Yaskawa INFORM job: DEMO_ROOF_UPPER_0625_3PAINT_63.JBI

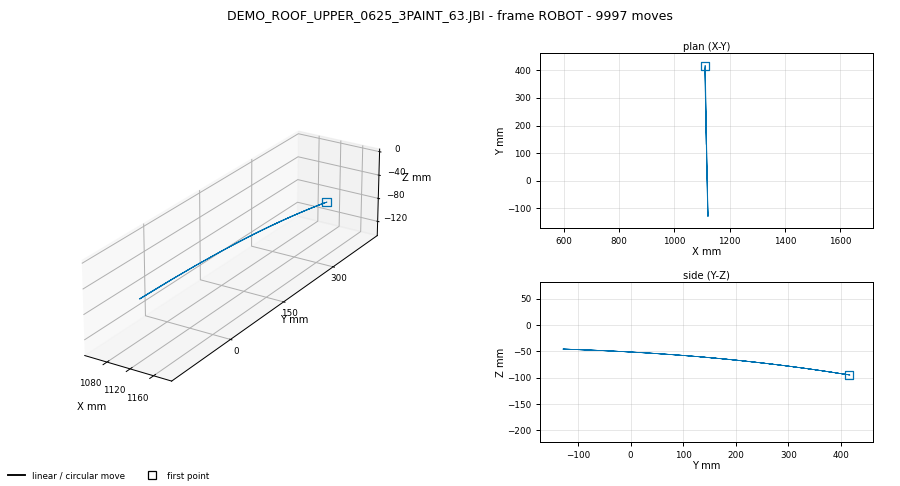
[picture p0: tool path of DEMO_ROOF_UPPER_0625_3PAINT_63.JBI in frame ROBOT, 9997 of 9997 moves have a stored position in this frame; points joined in program order, loops and branches not executed]
/JOB
//NAME DEMO_ROOF_UPPER_0625_3PAINT63
//POS
///NPOS 9997,0,0,0,0,0
///TOOL 0
///USER 0
///POSTYPE ROBOT
///RECTAN
///RCONF 1,0,0,0,0,0,0,0,0,0,0,0,0,0,0,0,0,0,0,0,0,0,0,0
C00000=1111.542,415.356,-94.503,-176.518,11.839,149.535
C00001=1111.541,415.109,-94.464,-176.519,11.832,149.534
C00002=1111.542,414.862,-94.424,-176.521,11.826,149.533
C00003=1111.542,414.615,-94.385,-176.522,11.820,149.532
C00004=1111.543,414.368,-94.345,-176.524,11.814,149.530
C00005=1111.545,414.121,-94.306,-176.526,11.807,149.529
C00006=1111.547,413.875,-94.266,-176.528,11.801,149.528
C00007=1111.549,413.627,-94.227,-176.529,11.795,149.527
C00008=1111.553,413.381,-94.187,-176.531,11.789,149.526
C00009=1111.556,413.135,-94.147,-176.533,11.783,149.525
C00010=1111.560,412.887,-94.107,-176.535,11.777,149.523
C00011=1111.563,412.640,-94.067,-176.536,11.771,149.522
C00012=1111.567,412.393,-94.027,-176.538,11.765,149.521
C00013=1111.570,412.147,-93.987,-176.540,11.759,149.520
C00014=1111.574,411.900,-93.948,-176.542,11.754,149.519
C00015=1111.577,411.654,-93.908,-176.543,11.747,149.518
C00016=1111.580,411.407,-93.869,-176.546,11.741,149.517
C00017=1111.584,411.160,-93.830,-176.547,11.736,149.516
C00018=1111.588,410.913,-93.789,-176.549,11.730,149.515
C00019=1111.591,410.666,-93.750,-176.551,11.725,149.514
C00020=1111.594,410.419,-93.710,-176.553,11.719,149.513
C00021=1111.598,410.172,-93.670,-176.554,11.713,149.512
C00022=1111.602,409.925,-93.631,-176.557,11.707,149.511
C00023=1111.605,409.679,-93.591,-176.559,11.703,149.510
C00024=1111.609,409.432,-93.552,-176.561,11.697,149.509
C00025=1111.612,409.185,-93.513,-176.562,11.691,149.508
C00026=1111.616,408.938,-93.473,-176.564,11.686,149.507
C00027=1111.619,408.692,-93.433,-176.567,11.680,149.506
C00028=1111.623,408.445,-93.394,-176.568,11.675,149.505
C00029=1111.626,408.198,-93.355,-176.570,11.670,149.504
C00030=1111.630,407.951,-93.316,-176.572,11.664,149.503
C00031=1111.633,407.704,-93.276,-176.574,11.659,149.503
C00032=1111.637,407.458,-93.236,-176.576,11.654,149.502
C00033=1111.641,407.211,-93.197,-176.578,11.649,149.501
C00034=1111.644,406.964,-93.158,-176.580,11.644,149.500
C00035=1111.648,406.717,-93.119,-176.582,11.639,149.499
C00036=1111.651,406.470,-93.079,-176.584,11.634,149.498
C00037=1111.654,406.223,-93.041,-176.586,11.629,149.498
C00038=1111.658,405.976,-93.002,-176.588,11.624,149.497
C00039=1111.662,405.729,-92.962,-176.590,11.619,149.496
C00040=1111.665,405.483,-92.922,-176.592,11.614,149.495
C00041=1111.668,405.236,-92.883,-176.594,11.609,149.494
C00042=1111.672,404.989,-92.844,-176.596,11.604,149.494
C00043=1111.676,404.742,-92.805,-176.599,11.599,149.493
C00044=1111.679,404.495,-92.765,-176.601,11.594,149.492
C00045=1111.682,404.248,-92.727,-176.603,11.590,149.492
C00046=1111.686,404.001,-92.687,-176.605,11.585,149.491
C00047=1111.690,403.754,-92.649,-176.607,11.581,149.490
C00048=1111.693,403.543,-92.615,-176.609,11.576,149.490
C00049=1111.696,403.331,-92.582,-176.611,11.572,149.489
C00050=1111.699,403.121,-92.548,-176.613,11.569,149.488
C00051=1111.702,402.909,-92.515,-176.615,11.565,149.488
C00052=1111.705,402.697,-92.482,-176.616,11.561,149.487
C00053=1111.708,402.486,-92.448,-176.619,11.556,149.487
C00054=1111.711,402.275,-92.415,-176.620,11.553,149.486
C00055=1111.714,402.063,-92.381,-176.622,11.549,149.486
C00056=1111.718,401.817,-92.342,-176.624,11.544,149.485
C00057=1111.721,401.570,-92.304,-176.626,11.541,149.484
C00058=1111.725,401.323,-92.264,-176.628,11.536,149.484
C00059=1111.729,401.075,-92.226,-176.631,11.532,149.483
C00060=1111.732,400.828,-92.187,-176.634,11.527,149.483
C00061=1111.735,400.582,-92.148,-176.635,11.523,149.482
C00062=1111.739,400.335,-92.109,-176.638,11.519,149.482
C00063=1111.743,400.087,-92.070,-176.640,11.514,149.481
C00064=1111.746,399.841,-92.032,-176.642,11.511,149.481
C00065=1111.750,399.594,-91.993,-176.645,11.506,149.480
C00066=1111.753,399.347,-91.953,-176.647,11.502,149.480
C00067=1111.757,399.100,-91.916,-176.649,11.498,149.479
C00068=1111.760,398.853,-91.876,-176.652,11.494,149.479
C00069=1111.764,398.606,-91.838,-176.654,11.490,149.478
C00070=1111.768,398.360,-91.799,-176.656,11.486,149.478
C00071=1111.771,398.113,-91.760,-176.658,11.482,149.477
C00072=1111.775,397.865,-91.722,-176.661,11.478,149.477
C00073=1111.778,397.618,-91.683,-176.663,11.475,149.477
C00074=1111.782,397.371,-91.644,-176.666,11.470,149.476
C00075=1111.786,397.125,-91.606,-176.668,11.467,149.476
C00076=1111.789,396.877,-91.568,-176.671,11.463,149.475
C00077=1111.793,396.630,-91.528,-176.673,11.459,149.475
C00078=1111.796,396.383,-91.490,-176.675,11.456,149.475
C00079=1111.800,396.137,-91.452,-176.678,11.451,149.474
C00080=1111.804,395.890,-91.414,-176.680,11.448,149.474
C00081=1111.807,395.643,-91.374,-176.682,11.444,149.473
C00082=1111.811,395.395,-91.336,-176.685,11.440,149.473
C00083=1111.815,395.149,-91.298,-176.687,11.437,149.473
C00084=1111.819,394.902,-91.259,-176.689,11.433,149.472
C00085=1111.821,394.655,-91.220,-176.692,11.430,149.472
C00086=1111.825,394.407,-91.182,-176.694,11.426,149.472
C00087=1111.829,394.161,-91.144,-176.697,11.423,149.472
C00088=1111.833,393.914,-91.105,-176.699,11.419,149.471
C00089=1111.836,393.666,-91.067,-176.702,11.416,149.471
C00090=1111.841,393.420,-91.029,-176.704,11.412,149.471
C00091=1111.843,393.173,-90.990,-176.707,11.409,149.471
C00092=1111.847,392.925,-90.952,-176.709,11.406,149.470
C00093=1111.851,392.679,-90.914,-176.711,11.402,149.470
C00094=1111.855,392.431,-90.876,-176.714,11.398,149.470
C00095=1111.858,392.185,-90.837,-176.717,11.395,149.470
C00096=1111.862,391.937,-90.798,-176.719,11.392,149.469
C00097=1111.866,391.690,-90.761,-176.722,11.389,149.469
C00098=1111.869,391.443,-90.723,-176.724,11.386,149.469
C00099=1111.872,391.196,-90.684,-176.727,11.383,149.469
C00100=1111.876,390.950,-90.646,-176.729,11.379,149.469
C00101=1111.880,390.702,-90.608,-176.732,11.376,149.468
C00102=1111.883,390.455,-90.570,-176.734,11.373,149.468
C00103=1111.887,390.208,-90.532,-176.737,11.370,149.468
C00104=1111.890,389.996,-90.499,-176.739,11.368,149.468
C00105=1111.893,389.786,-90.466,-176.742,11.365,149.468
C00106=1111.897,389.573,-90.434,-176.744,11.363,149.468
C00107=1111.899,389.362,-90.401,-176.746,11.359,149.468
C00108=1111.903,389.151,-90.368,-176.748,11.357,149.468
C00109=1111.906,388.939,-90.336,-176.750,11.355,149.468
C00110=1111.910,388.728,-90.303,-176.753,11.352,149.467
C00111=1111.912,388.517,-90.271,-176.755,11.349,149.467
C00112=1111.915,388.269,-90.233,-176.757,11.347,149.467
C00113=1111.920,388.022,-90.194,-176.760,11.344,149.467
C00114=1111.923,387.775,-90.156,-176.762,11.341,149.467
C00115=1111.927,387.529,-90.119,-176.765,11.339,149.467
C00116=1111.931,387.281,-90.080,-176.768,11.336,149.467
C00117=1111.934,387.034,-90.042,-176.770,11.333,149.467
C00118=1111.938,386.787,-90.005,-176.773,11.330,149.467
C00119=1111.941,386.540,-89.967,-176.775,11.328,149.467
C00120=1111.945,386.293,-89.929,-176.778,11.325,149.467
C00121=1111.949,386.045,-89.892,-176.781,11.322,149.467
C00122=1111.953,385.799,-89.854,-176.784,11.319,149.467
C00123=1111.956,385.551,-89.816,-176.786,11.317,149.467
C00124=1111.960,385.304,-89.777,-176.789,11.314,149.467
C00125=1111.963,385.057,-89.740,-176.792,11.311,149.467
C00126=1111.967,384.810,-89.702,-176.794,11.309,149.467
C00127=1111.970,384.563,-89.664,-176.797,11.306,149.467
C00128=1111.974,384.316,-89.626,-176.800,11.303,149.467
C00129=1111.978,384.069,-89.589,-176.802,11.301,149.467
C00130=1111.982,383.821,-89.551,-176.805,11.299,149.467
C00131=1111.985,383.575,-89.513,-176.808,11.296,149.467
C00132=1111.989,383.327,-89.476,-176.810,11.294,149.467
C00133=1111.992,383.081,-89.438,-176.814,11.290,149.467
C00134=1111.996,382.833,-89.401,-176.817,11.288,149.467
C00135=1112.000,382.586,-89.363,-176.820,11.285,149.467
C00136=1112.004,382.339,-89.325,-176.823,11.283,149.467
C00137=1112.008,382.092,-89.288,-176.827,11.280,149.468
C00138=1112.011,381.844,-89.250,-176.830,11.278,149.468
C00139=1112.015,381.598,-89.212,-176.833,11.275,149.468
C00140=1112.018,381.350,-89.175,-176.836,11.272,149.468
C00141=1112.022,381.103,-89.137,-176.840,11.269,149.468
C00142=1112.026,380.857,-89.100,-176.843,11.266,149.468
C00143=1112.029,380.609,-89.063,-176.846,11.264,149.468
C00144=1112.034,380.362,-89.024,-176.850,11.261,149.469
C00145=1112.037,380.115,-88.987,-176.853,11.259,149.469
C00146=1112.041,379.868,-88.950,-176.856,11.256,149.469
C00147=1112.044,379.620,-88.912,-176.859,11.253,149.469
C00148=1112.048,379.373,-88.875,-176.862,11.251,149.469
C00149=1112.052,379.127,-88.837,-176.866,11.249,149.469
C00150=1112.056,378.879,-88.800,-176.869,11.246,149.469
C00151=1112.059,378.632,-88.763,-176.872,11.242,149.470
C00152=1112.063,378.384,-88.725,-176.876,11.240,149.470
C00153=1112.067,378.138,-88.688,-176.879,11.237,149.470
C00154=1112.071,377.890,-88.651,-176.882,11.235,149.470
C00155=1112.074,377.643,-88.613,-176.886,11.232,149.470
C00156=1112.078,377.396,-88.576,-176.889,11.230,149.471
C00157=1112.082,377.149,-88.539,-176.892,11.228,149.471
C00158=1112.085,376.901,-88.501,-176.895,11.225,149.471
C00159=1112.089,376.654,-88.464,-176.898,11.222,149.471
C00160=1112.092,376.442,-88.432,-176.902,11.220,149.471
C00161=1112.095,376.231,-88.401,-176.904,11.218,149.471
C00162=1112.099,376.020,-88.369,-176.907,11.216,149.471
C00163=1112.102,375.808,-88.337,-176.910,11.214,149.472
C00164=1112.105,375.596,-88.306,-176.913,11.212,149.472
C00165=1112.108,375.385,-88.274,-176.915,11.209,149.472
C00166=1112.111,375.173,-88.242,-176.918,11.207,149.472
C00167=1112.114,374.962,-88.210,-176.921,11.205,149.472
C00168=1112.118,374.714,-88.173,-176.925,11.202,149.473
C00169=1112.122,374.467,-88.136,-176.928,11.200,149.473
C00170=1112.126,374.220,-88.099,-176.931,11.197,149.473
C00171=1112.130,373.973,-88.062,-176.935,11.195,149.473
C00172=1112.133,373.725,-88.025,-176.938,11.192,149.473
C00173=1112.137,373.478,-87.988,-176.941,11.190,149.474
C00174=1112.141,373.231,-87.951,-176.945,11.187,149.474
C00175=1112.144,372.983,-87.914,-176.948,11.185,149.474
C00176=1112.148,372.736,-87.877,-176.951,11.183,149.474
C00177=1112.152,372.489,-87.840,-176.954,11.180,149.474
C00178=1112.155,372.242,-87.804,-176.958,11.178,149.475
C00179=1112.159,371.994,-87.766,-176.961,11.175,149.475
C00180=1112.163,371.747,-87.729,-176.964,11.173,149.475
C00181=1112.167,371.500,-87.693,-176.968,11.170,149.475
C00182=1112.171,371.253,-87.656,-176.971,11.168,149.475
C00183=1112.174,371.005,-87.619,-176.975,11.165,149.476
C00184=1112.178,370.758,-87.582,-176.978,11.163,149.476
C00185=1112.182,370.511,-87.545,-176.981,11.161,149.476
C00186=1112.186,370.264,-87.509,-176.984,11.158,149.476
C00187=1112.190,370.017,-87.472,-176.988,11.156,149.477
C00188=1112.193,369.769,-87.435,-176.991,11.153,149.477
C00189=1112.196,369.522,-87.399,-176.994,11.151,149.477
C00190=1112.201,369.275,-87.362,-176.998,11.148,149.477
C00191=1112.205,369.028,-87.325,-177.001,11.146,149.478
C00192=1112.208,368.781,-87.289,-177.005,11.144,149.478
C00193=1112.212,368.533,-87.252,-177.008,11.141,149.478
C00194=1112.216,368.286,-87.215,-177.011,11.139,149.478
C00195=1112.219,368.038,-87.179,-177.015,11.136,149.478
C00196=1112.223,367.791,-87.142,-177.018,11.134,149.479
C00197=1112.227,367.544,-87.106,-177.022,11.131,149.479
C00198=1112.231,367.297,-87.069,-177.025,11.129,149.479
C00199=1112.235,367.050,-87.032,-177.028,11.127,149.480
C00200=1112.238,366.802,-86.996,-177.031,11.124,149.480
C00201=1112.242,366.554,-86.960,-177.035,11.122,149.480
C00202=1112.245,366.307,-86.923,-177.038,11.119,149.480
C00203=1112.250,366.060,-86.886,-177.042,11.117,149.481
C00204=1112.253,365.813,-86.851,-177.045,11.114,149.481
C00205=1112.257,365.566,-86.814,-177.048,11.112,149.481
C00206=1112.261,365.319,-86.778,-177.052,11.110,149.481
C00207=1112.265,365.071,-86.742,-177.055,11.107,149.482
C00208=1112.269,364.824,-86.705,-177.059,11.105,149.482
C00209=1112.272,364.576,-86.668,-177.062,11.102,149.482
C00210=1112.276,364.328,-86.632,-177.065,11.100,149.482
C00211=1112.280,364.081,-86.596,-177.069,11.097,149.482
C00212=1112.283,363.835,-86.559,-177.072,11.095,149.483
C00213=1112.287,363.587,-86.523,-177.075,11.094,149.483
C00214=1112.291,363.340,-86.487,-177.078,11.091,149.483
C00215=1112.295,363.092,-86.451,-177.082,11.089,149.483
C00216=1112.298,362.881,-86.420,-177.085,11.086,149.484
C00217=1112.301,362.669,-86.389,-177.088,11.085,149.484
C00218=1112.304,362.456,-86.358,-177.091,11.082,149.484
C00219=1112.307,362.245,-86.327,-177.094,11.080,149.484
C00220=1112.311,362.034,-86.296,-177.096,11.079,149.485
C00221=1112.314,361.822,-86.265,-177.100,11.076,149.485
C00222=1112.318,361.610,-86.234,-177.102,11.075,149.485
C00223=1112.321,361.398,-86.204,-177.105,11.072,149.485
C00224=1112.325,361.151,-86.167,-177.109,11.070,149.486
C00225=1112.329,360.903,-86.131,-177.112,11.067,149.486
C00226=1112.332,360.656,-86.095,-177.115,11.065,149.486
C00227=1112.336,360.409,-86.059,-177.119,11.062,149.486
C00228=1112.340,360.161,-86.023,-177.122,11.060,149.486
C00229=1112.343,359.914,-85.987,-177.126,11.058,149.487
C00230=1112.348,359.666,-85.951,-177.129,11.055,149.487
C00231=1112.351,359.419,-85.915,-177.132,11.053,149.487
C00232=1112.355,359.172,-85.879,-177.135,11.051,149.488
C00233=1112.359,358.925,-85.844,-177.138,11.048,149.488
C00234=1112.363,358.677,-85.807,-177.142,11.046,149.488
C00235=1112.366,358.430,-85.771,-177.145,11.044,149.488
C00236=1112.370,358.182,-85.736,-177.149,11.041,149.489
C00237=1112.374,357.935,-85.700,-177.152,11.039,149.489
C00238=1112.378,357.687,-85.664,-177.155,11.036,149.489
C00239=1112.381,357.440,-85.628,-177.159,11.034,149.489
C00240=1112.385,357.193,-85.592,-177.162,11.032,149.490
C00241=1112.389,356.945,-85.557,-177.166,11.029,149.490
C00242=1112.393,356.697,-85.520,-177.169,11.027,149.490
C00243=1112.397,356.450,-85.485,-177.172,11.024,149.490
C00244=1112.400,356.203,-85.449,-177.175,11.022,149.491
C00245=1112.404,355.956,-85.413,-177.179,11.020,149.491
C00246=1112.408,355.709,-85.378,-177.182,11.017,149.491
C00247=1112.412,355.461,-85.342,-177.186,11.015,149.491
C00248=1112.416,355.213,-85.306,-177.189,11.012,149.492
C00249=1112.420,354.966,-85.271,-177.192,11.010,149.492
C00250=1112.423,354.718,-85.235,-177.196,11.008,149.492
C00251=1112.427,354.471,-85.199,-177.199,11.005,149.492
C00252=1112.431,354.223,-85.164,-177.202,11.003,149.492
C00253=1112.435,353.977,-85.129,-177.206,11.000,149.493
C00254=1112.439,353.729,-85.093,-177.209,10.998,149.493
C00255=1112.442,353.482,-85.058,-177.213,10.996,149.493
C00256=1112.447,353.234,-85.022,-177.216,10.993,149.494
C00257=1112.450,352.986,-84.986,-177.219,10.991,149.494
C00258=1112.454,352.739,-84.950,-177.223,10.987,149.494
C00259=1112.458,352.492,-84.915,-177.227,10.985,149.494
C00260=1112.462,352.244,-84.880,-177.230,10.982,149.494
C00261=1112.466,351.997,-84.844,-177.233,10.980,149.495
C00262=1112.469,351.749,-84.809,-177.236,10.978,149.495
C00263=1112.473,351.501,-84.774,-177.240,10.975,149.495
C00264=1112.478,351.255,-84.739,-177.243,10.973,149.495
C00265=1112.481,351.007,-84.703,-177.246,10.970,149.496
C00266=1112.485,350.760,-84.667,-177.250,10.968,149.496
C00267=1112.489,350.512,-84.632,-177.253,10.965,149.496
C00268=1112.492,350.264,-84.597,-177.256,10.963,149.496
C00269=1112.497,350.017,-84.562,-177.260,10.960,149.496
C00270=1112.500,349.770,-84.526,-177.263,10.958,149.497
C00271=1112.504,349.522,-84.491,-177.266,10.955,149.497
C00272=1112.507,349.310,-84.461,-177.269,10.954,149.497
C00273=1112.511,349.098,-84.430,-177.272,10.951,149.497
C00274=1112.514,348.886,-84.401,-177.275,10.949,149.497
C00275=1112.518,348.675,-84.371,-177.277,10.948,149.498
C00276=1112.521,348.462,-84.341,-177.280,10.945,149.498
C00277=1112.525,348.251,-84.310,-177.283,10.943,149.498
C00278=1112.528,348.038,-84.281,-177.285,10.941,149.498
C00279=1112.531,347.827,-84.250,-177.288,10.939,149.498
C00280=1112.534,347.579,-84.215,-177.292,10.936,149.499
C00281=1112.538,347.331,-84.180,-177.295,10.934,149.499
C00282=1112.543,347.084,-84.145,-177.298,10.931,149.499
C00283=1112.547,346.836,-84.110,-177.301,10.929,149.499
C00284=1112.550,346.589,-84.074,-177.304,10.927,149.499
C00285=1112.555,346.341,-84.040,-177.307,10.924,149.500
C00286=1112.558,346.094,-84.005,-177.311,10.922,149.500
C00287=1112.561,345.847,-83.969,-177.314,10.919,149.500
C00288=1112.566,345.599,-83.935,-177.317,10.917,149.500
C00289=1112.570,345.352,-83.899,-177.320,10.914,149.500
C00290=1112.574,345.103,-83.865,-177.323,10.912,149.500
C00291=1112.578,344.856,-83.830,-177.327,10.909,149.501
C00292=1112.581,344.609,-83.795,-177.330,10.907,149.501
C00293=1112.586,344.361,-83.761,-177.332,10.905,149.501
C00294=1112.589,344.114,-83.725,-177.336,10.902,149.501
C00295=1112.593,343.866,-83.690,-177.339,10.900,149.501
C00296=1112.597,343.619,-83.656,-177.342,10.897,149.502
C00297=1112.601,343.371,-83.621,-177.346,10.895,149.502
C00298=1112.605,343.124,-83.586,-177.348,10.892,149.502
C00299=1112.609,342.876,-83.551,-177.352,10.890,149.502
C00300=1112.612,342.628,-83.517,-177.355,10.887,149.502
C00301=1112.617,342.381,-83.482,-177.358,10.885,149.503
C00302=1112.620,342.134,-83.447,-177.362,10.882,149.503
C00303=1112.625,341.886,-83.412,-177.365,10.879,149.503
C00304=1112.628,341.638,-83.378,-177.367,10.878,149.503
C00305=1112.633,341.391,-83.343,-177.371,10.875,149.503
C00306=1112.636,341.143,-83.308,-177.374,10.873,149.504
C00307=1112.640,340.896,-83.274,-177.377,10.870,149.504
C00308=1112.644,340.648,-83.239,-177.380,10.868,149.504
C00309=1112.648,340.400,-83.204,-177.384,10.865,149.504
C00310=1112.652,340.154,-83.170,-177.387,10.863,149.504
C00311=1112.656,339.905,-83.135,-177.390,10.860,149.505
C00312=1112.660,339.658,-83.101,-177.393,10.857,149.505
C00313=1112.664,339.410,-83.066,-177.396,10.855,149.505
C00314=1112.668,339.163,-83.032,-177.399,10.853,149.505
C00315=1112.671,338.915,-82.998,-177.402,10.851,149.505
C00316=1112.676,338.668,-82.963,-177.405,10.848,149.506
C00317=1112.680,338.419,-82.928,-177.409,10.846,149.506
C00318=1112.683,338.173,-82.894,-177.412,10.843,149.506
C00319=1112.687,337.925,-82.859,-177.415,10.841,149.506
C00320=1112.691,337.678,-82.825,-177.418,10.838,149.506
C00321=1112.695,337.430,-82.790,-177.421,10.836,149.506
C00322=1112.699,337.183,-82.756,-177.425,10.833,149.507
C00323=1112.703,336.934,-82.721,-177.428,10.831,149.507
C00324=1112.707,336.687,-82.688,-177.431,10.828,149.507
C00325=1112.711,336.439,-82.653,-177.434,10.826,149.507
C00326=1112.715,336.192,-82.619,-177.437,10.824,149.508
C00327=1112.719,335.945,-82.584,-177.440,10.821,149.508
C00328=1112.722,335.732,-82.555,-177.443,10.818,149.508
C00329=1112.726,335.519,-82.526,-177.446,10.817,149.508
C00330=1112.729,335.307,-82.496,-177.448,10.815,149.508
C00331=1112.732,335.096,-82.468,-177.452,10.812,149.508
C00332=1112.735,334.884,-82.438,-177.454,10.810,149.508
C00333=1112.739,334.672,-82.408,-177.457,10.809,149.509
C00334=1112.742,334.460,-82.379,-177.459,10.806,149.509
C00335=1112.746,334.247,-82.350,-177.462,10.804,149.509
C00336=1112.750,334.000,-82.317,-177.465,10.801,149.509
C00337=1112.754,333.752,-82.282,-177.468,10.799,149.509
C00338=1112.758,333.505,-82.248,-177.472,10.796,149.510
C00339=1112.762,333.257,-82.213,-177.475,10.794,149.510
C00340=1112.765,333.010,-82.179,-177.478,10.791,149.510
C00341=1112.769,332.762,-82.146,-177.481,10.790,149.510
C00342=1112.773,332.514,-82.111,-177.484,10.787,149.510
C00343=1112.777,332.267,-82.077,-177.487,10.784,149.510
C00344=1112.781,332.019,-82.043,-177.490,10.782,149.511
C00345=1112.785,331.771,-82.009,-177.494,10.779,149.511
C00346=1112.789,331.524,-81.975,-177.496,10.777,149.511
C00347=1112.792,331.276,-81.941,-177.500,10.774,149.511
C00348=1112.797,331.028,-81.907,-177.503,10.772,149.511
C00349=1112.801,330.781,-81.874,-177.506,10.769,149.512
C00350=1112.804,330.533,-81.839,-177.509,10.767,149.512
C00351=1112.809,330.285,-81.806,-177.513,10.764,149.512
C00352=1112.813,330.038,-81.772,-177.515,10.762,149.512
C00353=1112.817,329.789,-81.738,-177.518,10.760,149.512
C00354=1112.820,329.542,-81.704,-177.522,10.757,149.513
C00355=1112.825,329.295,-81.670,-177.525,10.755,149.513
C00356=1112.829,329.046,-81.636,-177.528,10.752,149.513
C00357=1112.832,328.799,-81.602,-177.531,10.750,149.513
C00358=1112.837,328.551,-81.569,-177.534,10.747,149.513
C00359=1112.840,328.304,-81.535,-177.537,10.744,149.513
C00360=1112.845,328.056,-81.501,-177.541,10.742,149.514
C00361=1112.848,327.808,-81.467,-177.544,10.739,149.514
C00362=1112.853,327.561,-81.434,-177.547,10.737,149.514
C00363=1112.856,327.313,-81.400,-177.550,10.735,149.514
C00364=1112.860,327.065,-81.367,-177.553,10.732,149.515
C00365=1112.865,326.818,-81.332,-177.556,10.730,149.515
C00366=1112.869,326.570,-81.299,-177.559,10.727,149.515
C00367=1112.872,326.322,-81.266,-177.563,10.725,149.515
C00368=1112.876,326.075,-81.232,-177.565,10.722,149.515
C00369=1112.880,325.827,-81.199,-177.569,10.720,149.515
C00370=1112.884,325.579,-81.166,-177.572,10.717,149.516
C00371=1112.888,325.332,-81.132,-177.575,10.714,149.516
C00372=1112.892,325.084,-81.098,-177.578,10.712,149.516
C00373=1112.897,324.835,-81.064,-177.581,10.710,149.516
C00374=1112.900,324.588,-81.030,-177.584,10.707,149.516
C00375=1112.905,324.341,-80.997,-177.587,10.705,149.517
C00376=1112.908,324.092,-80.964,-177.591,10.703,149.517
C00377=1112.912,323.845,-80.930,-177.593,10.700,149.517
C00378=1112.916,323.597,-80.897,-177.597,10.697,149.517
C00379=1112.920,323.350,-80.864,-177.600,10.695,149.517
C00380=1112.924,323.102,-80.830,-177.603,10.692,149.517
C00381=1112.928,322.854,-80.797,-177.606,10.690,149.518
C00382=1112.932,322.606,-80.763,-177.609,10.687,149.518
C00383=1112.936,322.359,-80.730,-177.613,10.684,149.518
C00384=1112.939,322.147,-80.702,-177.615,10.682,149.518
C00385=1112.943,321.934,-80.673,-177.618,10.681,149.518
C00386=1112.946,321.722,-80.645,-177.621,10.678,149.518
C00387=1112.949,321.510,-80.616,-177.623,10.676,149.519
C00388=1112.953,321.298,-80.588,-177.626,10.674,149.519
C00389=1112.956,321.085,-80.559,-177.628,10.672,149.519
C00390=1112.960,320.873,-80.531,-177.631,10.670,149.519
C00391=1112.963,320.660,-80.502,-177.633,10.668,149.519
C00392=1112.967,320.413,-80.469,-177.637,10.665,149.519
C00393=1112.971,320.165,-80.436,-177.640,10.663,149.520
C00394=1112.975,319.917,-80.403,-177.643,10.660,149.520
C00395=1112.979,319.670,-80.370,-177.646,10.658,149.520
C00396=1112.983,319.422,-80.337,-177.649,10.655,149.520
C00397=1112.987,319.174,-80.304,-177.653,10.653,149.520
C00398=1112.991,318.927,-80.270,-177.656,10.650,149.521
C00399=1112.995,318.678,-80.237,-177.659,10.647,149.521
C00400=1112.999,318.430,-80.204,-177.662,10.646,149.521
C00401=1113.002,318.183,-80.171,-177.664,10.643,149.521
C00402=1113.007,317.935,-80.138,-177.668,10.640,149.521
C00403=1113.011,317.688,-80.105,-177.671,10.638,149.521
C00404=1113.015,317.440,-80.072,-177.674,10.635,149.522
C00405=1113.019,317.192,-80.039,-177.677,10.633,149.522
C00406=1113.023,316.944,-80.005,-177.680,10.630,149.522
C00407=1113.027,316.697,-79.973,-177.684,10.628,149.522
C00408=1113.031,316.449,-79.940,-177.687,10.625,149.522
C00409=1113.035,316.201,-79.907,-177.690,10.622,149.522
C00410=1113.039,315.953,-79.874,-177.693,10.621,149.523
C00411=1113.043,315.706,-79.842,-177.695,10.618,149.523
C00412=1113.047,315.458,-79.808,-177.699,10.615,149.523
C00413=1113.051,315.210,-79.776,-177.702,10.613,149.523
C00414=1113.055,314.962,-79.743,-177.705,10.610,149.523
C00415=1113.059,314.714,-79.710,-177.708,10.608,149.524
C00416=1113.063,314.467,-79.677,-177.711,10.605,149.524
C00417=1113.067,314.218,-79.645,-177.715,10.603,149.524
C00418=1113.072,313.971,-79.612,-177.718,10.600,149.524
C00419=1113.075,313.723,-79.579,-177.721,10.597,149.524
C00420=1113.079,313.475,-79.547,-177.724,10.596,149.525
C00421=1113.083,313.227,-79.513,-177.727,10.593,149.525
C00422=1113.087,312.980,-79.481,-177.730,10.591,149.525
C00423=1113.091,312.731,-79.448,-177.733,10.588,149.525
C00424=1113.095,312.484,-79.415,-177.736,10.585,149.525
C00425=1113.099,312.236,-79.383,-177.739,10.583,149.525
C00426=1113.103,311.988,-79.350,-177.742,10.580,149.526
C00427=1113.107,311.740,-79.318,-177.746,10.578,149.526
C00428=1113.111,311.492,-79.285,-177.749,10.575,149.526
C00429=1113.115,311.244,-79.252,-177.752,10.572,149.526
C00430=1113.119,310.996,-79.220,-177.755,10.570,149.526
C00431=1113.124,310.749,-79.187,-177.758,10.568,149.526
C00432=1113.127,310.501,-79.156,-177.760,10.565,149.527
C00433=1113.132,310.254,-79.122,-177.764,10.563,149.527
C00434=1113.136,310.005,-79.090,-177.767,10.560,149.527
C00435=1113.139,309.758,-79.057,-177.770,10.558,149.527
C00436=1113.144,309.509,-79.025,-177.773,10.555,149.527
C00437=1113.147,309.262,-78.992,-177.776,10.552,149.527
C00438=1113.152,309.014,-78.960,-177.780,10.550,149.528
C00439=1113.155,308.766,-78.928,-177.783,10.547,149.528
C00440=1113.159,308.554,-78.900,-177.785,10.546,149.528
C00441=1113.163,308.341,-78.872,-177.788,10.544,149.528
C00442=1113.167,308.129,-78.844,-177.791,10.541,149.528
C00443=1113.170,307.917,-78.817,-177.793,10.539,149.529
C00444=1113.173,307.704,-78.789,-177.796,10.537,149.529
C00445=1113.177,307.492,-78.762,-177.798,10.534,149.529
C00446=1113.180,307.280,-78.734,-177.801,10.533,149.529
C00447=1113.184,307.067,-78.707,-177.803,10.531,149.529
C00448=1113.188,306.820,-78.674,-177.806,10.528,149.529
C00449=1113.192,306.572,-78.642,-177.810,10.525,149.529
C00450=1113.196,306.323,-78.609,-177.813,10.523,149.530
C00451=1113.200,306.075,-78.577,-177.816,10.520,149.530
C00452=1113.204,305.828,-78.545,-177.819,10.518,149.530
C00453=1113.208,305.580,-78.513,-177.822,10.515,149.530
C00454=1113.212,305.332,-78.481,-177.826,10.513,149.530
C00455=1113.216,305.084,-78.448,-177.828,10.510,149.530
C00456=1113.220,304.836,-78.417,-177.831,10.508,149.531
C00457=1113.224,304.589,-78.384,-177.834,10.505,149.531
C00458=1113.229,304.341,-78.352,-177.837,10.503,149.531
C00459=1113.232,304.093,-78.320,-177.840,10.500,149.531
C00460=1113.237,303.844,-78.288,-177.844,10.498,149.531
C00461=1113.241,303.597,-78.256,-177.847,10.495,149.531
C00462=1113.245,303.349,-78.224,-177.850,10.493,149.532
C00463=1113.249,303.100,-78.192,-177.853,10.490,149.532
C00464=1113.253,302.852,-78.160,-177.856,10.487,149.532
C00465=1113.257,302.605,-78.129,-177.859,10.485,149.532
C00466=1113.262,302.357,-78.096,-177.862,10.483,149.532
C00467=1113.265,302.109,-78.064,-177.865,10.480,149.533
C00468=1113.270,301.861,-78.033,-177.868,10.478,149.533
C00469=1113.274,301.613,-78.000,-177.871,10.475,149.533
C00470=1113.278,301.365,-77.969,-177.874,10.473,149.533
C00471=1113.282,301.118,-77.937,-177.877,10.470,149.533
C00472=1113.286,300.870,-77.905,-177.881,10.467,149.534
C00473=1113.290,300.621,-77.873,-177.884,10.465,149.534
C00474=1113.294,300.373,-77.841,-177.887,10.462,149.534
C00475=1113.298,300.126,-77.809,-177.889,10.460,149.534
C00476=1113.302,299.878,-77.778,-177.893,10.458,149.534
C00477=1113.306,299.629,-77.745,-177.895,10.455,149.534
C00478=1113.311,299.382,-77.714,-177.899,10.453,149.535
C00479=1113.314,299.134,-77.682,-177.902,10.450,149.535
C00480=1113.319,298.886,-77.651,-177.905,10.447,149.535
C00481=1113.323,298.638,-77.619,-177.908,10.445,149.535
C00482=1113.326,298.390,-77.587,-177.911,10.442,149.535
C00483=1113.332,298.142,-77.555,-177.914,10.439,149.535
C00484=1113.335,297.894,-77.523,-177.918,10.437,149.536
C00485=1113.339,297.646,-77.492,-177.920,10.435,149.536
C00486=1113.344,297.398,-77.461,-177.923,10.433,149.536
C00487=1113.347,297.150,-77.429,-177.926,10.430,149.536
C00488=1113.351,296.902,-77.397,-177.930,10.427,149.536
C00489=1113.356,296.654,-77.366,-177.932,10.425,149.536
C00490=1113.359,296.406,-77.335,-177.936,10.422,149.537
C00491=1113.364,296.159,-77.303,-177.939,10.419,149.537
C00492=1113.368,295.910,-77.271,-177.942,10.417,149.537
C00493=1113.373,295.663,-77.240,-177.945,10.414,149.537
C00494=1113.376,295.415,-77.208,-177.948,10.413,149.537
C00495=1113.380,295.166,-77.177,-177.951,10.410,149.538
C00496=1113.383,294.954,-77.150,-177.954,10.407,149.538
C00497=1113.387,294.741,-77.123,-177.956,10.405,149.538
C00498=1113.391,294.529,-77.096,-177.959,10.403,149.538
C00499=1113.394,294.316,-77.069,-177.961,10.401,149.538
C00500=1113.397,294.104,-77.042,-177.964,10.399,149.538
C00501=1113.401,293.891,-77.016,-177.966,10.397,149.538
C00502=1113.405,293.679,-76.988,-177.969,10.394,149.539
C00503=1113.408,293.466,-76.962,-177.972,10.392,149.539
C00504=1113.413,293.218,-76.931,-177.975,10.390,149.539
C00505=1113.416,292.970,-76.899,-177.978,10.387,149.539
C00506=1113.420,292.722,-76.868,-177.981,10.384,149.539
C00507=1113.425,292.474,-76.837,-177.984,10.382,149.539
C00508=1113.429,292.226,-76.805,-177.987,10.380,149.540
C00509=1113.433,291.978,-76.774,-177.990,10.377,149.540
C00510=1113.437,291.730,-76.743,-177.993,10.375,149.540
C00511=1113.441,291.482,-76.711,-177.996,10.372,149.540
C00512=1113.445,291.234,-76.680,-177.999,10.369,149.540
C00513=1113.449,290.987,-76.649,-178.002,10.367,149.541
C00514=1113.453,290.738,-76.618,-178.005,10.364,149.541
C00515=1113.457,290.490,-76.587,-178.009,10.362,149.541
C00516=1113.462,290.243,-76.556,-178.012,10.359,149.541
C00517=1113.466,289.994,-76.525,-178.014,10.357,149.541
C00518=1113.470,289.746,-76.494,-178.017,10.355,149.541
C00519=1113.474,289.498,-76.462,-178.020,10.352,149.541
C00520=1113.478,289.250,-76.432,-178.024,10.349,149.542
C00521=1113.482,289.002,-76.401,-178.026,10.347,149.542
C00522=1113.486,288.754,-76.369,-178.030,10.344,149.542
C00523=1113.490,288.506,-76.338,-178.033,10.342,149.542
C00524=1113.495,288.258,-76.308,-178.036,10.339,149.542
C00525=1113.499,288.010,-76.277,-178.039,10.336,149.543
C00526=1113.503,287.762,-76.246,-178.041,10.334,149.543
C00527=1113.507,287.514,-76.215,-178.045,10.332,149.543
C00528=1113.511,287.266,-76.184,-178.048,10.329,149.543
C00529=1113.516,287.018,-76.153,-178.051,10.327,149.543
C00530=1113.520,286.770,-76.123,-178.054,10.324,149.543
C00531=1113.524,286.521,-76.092,-178.057,10.322,149.544
C00532=1113.528,286.274,-76.060,-178.060,10.319,149.544
C00533=1113.531,286.026,-76.030,-178.063,10.316,149.544
C00534=1113.536,285.778,-75.999,-178.066,10.314,149.544
C00535=1113.540,285.530,-75.968,-178.069,10.312,149.544
C00536=1113.544,285.281,-75.937,-178.072,10.309,149.544
C00537=1113.548,285.033,-75.907,-178.075,10.306,149.545
C00538=1113.553,284.785,-75.876,-178.078,10.304,149.545
C00539=1113.557,284.537,-75.845,-178.081,10.301,149.545
C00540=1113.561,284.289,-75.815,-178.084,10.298,149.545
C00541=1113.565,284.041,-75.784,-178.088,10.296,149.545
C00542=1113.569,283.792,-75.753,-178.091,10.293,149.545
C00543=1113.573,283.545,-75.723,-178.093,10.292,149.546
C00544=1113.578,283.297,-75.692,-178.096,10.289,149.546
C00545=1113.582,283.048,-75.661,-178.100,10.286,149.546
C00546=1113.586,282.801,-75.631,-178.102,10.284,149.546
C00547=1113.590,282.553,-75.600,-178.105,10.281,149.546
C00548=1113.594,282.304,-75.569,-178.109,10.279,149.547
C00549=1113.598,282.056,-75.538,-178.112,10.276,149.547
C00550=1113.603,281.808,-75.508,-178.115,10.273,149.547
C00551=1113.607,281.560,-75.478,-178.118,10.271,149.547
C00552=1113.610,281.348,-75.452,-178.120,10.269,149.547
C00553=1113.614,281.135,-75.425,-178.123,10.267,149.547
C00554=1113.617,280.922,-75.399,-178.126,10.264,149.548
C00555=1113.621,280.709,-75.373,-178.128,10.262,149.548
C00556=1113.625,280.497,-75.347,-178.131,10.259,149.548
C00557=1113.628,280.284,-75.321,-178.133,10.257,149.548
C00558=1113.632,280.071,-75.295,-178.137,10.255,149.548
C00559=1113.636,279.858,-75.269,-178.139,10.253,149.548
C00560=1113.640,279.611,-75.239,-178.142,10.250,149.548
C00561=1113.644,279.363,-75.208,-178.145,10.248,149.549
C00562=1113.648,279.115,-75.178,-178.148,10.245,149.549
C00563=1113.652,278.866,-75.147,-178.151,10.242,149.549
C00564=1113.656,278.618,-75.117,-178.155,10.240,149.549
C00565=1113.661,278.370,-75.086,-178.158,10.237,149.549
C00566=1113.665,278.122,-75.056,-178.160,10.234,149.549
C00567=1113.669,277.874,-75.027,-178.163,10.232,149.549
C00568=1113.673,277.625,-74.996,-178.167,10.229,149.550
C00569=1113.677,277.377,-74.966,-178.170,10.226,149.550
C00570=1113.682,277.129,-74.936,-178.173,10.224,149.550
C00571=1113.686,276.882,-74.905,-178.176,10.221,149.550
C00572=1113.690,276.633,-74.876,-178.179,10.219,149.550
C00573=1113.694,276.385,-74.845,-178.181,10.217,149.550
C00574=1113.698,276.136,-74.815,-178.184,10.214,149.550
C00575=1113.702,275.889,-74.785,-178.187,10.211,149.551
C00576=1113.706,275.641,-74.754,-178.190,10.208,149.551
C00577=1113.711,275.393,-74.725,-178.193,10.206,149.551
C00578=1113.715,275.145,-74.695,-178.196,10.203,149.551
C00579=1113.719,274.896,-74.664,-178.199,10.200,149.551
C00580=1113.723,274.648,-74.634,-178.202,10.198,149.551
C00581=1113.727,274.400,-74.605,-178.205,10.195,149.551
C00582=1113.732,274.152,-74.574,-178.208,10.192,149.551
C00583=1113.736,273.903,-74.544,-178.211,10.189,149.552
C00584=1113.740,273.655,-74.515,-178.214,10.188,149.552
C00585=1113.744,273.408,-74.485,-178.217,10.185,149.552
C00586=1113.749,273.159,-74.455,-178.220,10.182,149.552
C00587=1113.753,272.911,-74.425,-178.222,10.179,149.552
C00588=1113.756,272.662,-74.395,-178.225,10.177,149.552
C00589=1113.760,272.414,-74.365,-178.228,10.174,149.552
C00590=1113.765,272.166,-74.335,-178.231,10.171,149.552
C00591=1113.769,271.918,-74.305,-178.234,10.168,149.553
C00592=1113.773,271.670,-74.276,-178.237,10.166,149.553
C00593=1113.777,271.422,-74.246,-178.239,10.164,149.553
C00594=1113.781,271.174,-74.216,-178.242,10.161,149.553
C00595=1113.786,270.925,-74.186,-178.245,10.158,149.553
C00596=1113.790,270.677,-74.156,-178.248,10.155,149.553
C00597=1113.794,270.429,-74.126,-178.251,10.153,149.553
C00598=1113.798,270.181,-74.097,-178.254,10.151,149.553
C00599=1113.803,269.933,-74.068,-178.256,10.148,149.553
C00600=1113.807,269.684,-74.038,-178.259,10.145,149.553
C00601=1113.811,269.436,-74.007,-178.262,10.142,149.554
C00602=1113.816,269.188,-73.978,-178.265,10.141,149.554
C00603=1113.820,268.940,-73.948,-178.268,10.138,149.554
C00604=1113.824,268.692,-73.919,-178.271,10.135,149.554
C00605=1113.828,268.443,-73.889,-178.274,10.132,149.554
C00606=1113.832,268.196,-73.859,-178.276,10.130,149.554
C00607=1113.836,267.947,-73.830,-178.279,10.128,149.554
C00608=1113.840,267.734,-73.805,-178.281,10.125,149.554
C00609=1113.844,267.522,-73.779,-178.284,10.123,149.554
C00610=1113.847,267.309,-73.754,-178.286,10.121,149.555
C00611=1113.851,267.096,-73.728,-178.289,10.119,149.555
C00612=1113.855,266.883,-73.703,-178.291,10.117,149.555
C00613=1113.858,266.670,-73.678,-178.293,10.115,149.555
C00614=1113.862,266.457,-73.653,-178.295,10.113,149.555
C00615=1113.866,266.244,-73.627,-178.298,10.110,149.555
C00616=1113.870,265.996,-73.598,-178.301,10.108,149.555
C00617=1113.874,265.748,-73.568,-178.304,10.105,149.555
C00618=1113.878,265.499,-73.539,-178.307,10.102,149.556
C00619=1113.883,265.252,-73.510,-178.309,10.100,149.556
C00620=1113.887,265.003,-73.480,-178.312,10.098,149.556
C00621=1113.891,264.755,-73.451,-178.315,10.095,149.556
C00622=1113.896,264.507,-73.422,-178.317,10.093,149.556
C00623=1113.900,264.259,-73.392,-178.320,10.090,149.556
C00624=1113.904,264.010,-73.363,-178.323,10.088,149.556
C00625=1113.908,263.762,-73.333,-178.327,10.084,149.556
C00626=1113.912,263.514,-73.304,-178.330,10.081,149.557
C00627=1113.916,263.266,-73.274,-178.333,10.079,149.557
C00628=1113.920,263.018,-73.245,-178.336,10.076,149.557
C00629=1113.925,262.769,-73.217,-178.339,10.073,149.557
C00630=1113.929,262.521,-73.188,-178.342,10.071,149.557
C00631=1113.933,262.273,-73.158,-178.345,10.068,149.557
C00632=1113.938,262.025,-73.129,-178.348,10.065,149.557
C00633=1113.942,261.776,-73.099,-178.351,10.062,149.557
C00634=1113.946,261.527,-73.071,-178.354,10.060,149.558
C00635=1113.950,261.279,-73.041,-178.357,10.057,149.558
C00636=1113.955,261.032,-73.012,-178.360,10.055,149.558
C00637=1113.959,260.784,-72.983,-178.364,10.051,149.558
C00638=1113.963,260.535,-72.954,-178.367,10.048,149.558
C00639=1113.967,260.287,-72.925,-178.370,10.045,149.558
C00640=1113.971,260.038,-72.895,-178.373,10.043,149.558
C00641=1113.977,259.790,-72.867,-178.375,10.040,149.559
C00642=1113.980,259.542,-72.838,-178.378,10.037,149.558
C00643=1113.984,259.294,-72.809,-178.381,10.034,149.559
C00644=1113.989,259.045,-72.780,-178.384,10.031,149.559
C00645=1113.993,258.797,-72.751,-178.387,10.029,149.559
C00646=1113.997,258.549,-72.722,-178.390,10.026,149.559
C00647=1114.001,258.301,-72.693,-178.393,10.023,149.559
C00648=1114.006,258.052,-72.664,-178.396,10.020,149.559
C00649=1114.010,257.803,-72.635,-178.398,10.018,149.559
C00650=1114.013,257.555,-72.606,-178.400,10.015,149.559
C00651=1114.019,257.307,-72.578,-178.403,10.012,149.559
C00652=1114.023,257.059,-72.548,-178.406,10.010,149.559
C00653=1114.026,256.810,-72.520,-178.409,10.007,149.559
C00654=1114.031,256.562,-72.491,-178.412,10.004,149.559
C00655=1114.036,256.314,-72.463,-178.415,10.001,149.559
C00656=1114.040,256.066,-72.433,-178.418,9.998,149.560
C00657=1114.044,255.817,-72.405,-178.420,9.996,149.559
C00658=1114.048,255.570,-72.376,-178.421,9.994,149.559
C00659=1114.053,255.321,-72.347,-178.423,9.992,149.559
C00660=1114.056,255.073,-72.318,-178.425,9.990,149.559
C00661=1114.061,254.824,-72.289,-178.426,9.988,149.559
C00662=1114.065,254.577,-72.261,-178.428,9.986,149.559
C00663=1114.069,254.328,-72.232,-178.430,9.984,149.559
C00664=1114.074,254.115,-72.207,-178.432,9.982,149.559
C00665=1114.076,253.902,-72.183,-178.434,9.980,149.559
C00666=1114.081,253.689,-72.159,-178.436,9.978,149.560
C00667=1114.084,253.476,-72.135,-178.438,9.976,149.560
C00668=1114.088,253.263,-72.109,-178.441,9.974,149.560
C00669=1114.091,253.050,-72.085,-178.442,9.972,149.560
C00670=1114.095,252.837,-72.060,-178.445,9.970,149.560
C00671=1114.098,252.625,-72.036,-178.447,9.968,149.560
C00672=1114.103,252.376,-72.007,-178.449,9.966,149.560
C00673=1114.108,252.127,-71.979,-178.453,9.964,149.560
C00674=1114.112,251.879,-71.950,-178.456,9.961,149.561
C00675=1114.116,251.631,-71.921,-178.459,9.958,149.561
C00676=1114.120,251.383,-71.893,-178.462,9.956,149.561
C00677=1114.125,251.134,-71.865,-178.465,9.953,149.561
C00678=1114.128,250.886,-71.836,-178.468,9.951,149.561
C00679=1114.133,250.638,-71.807,-178.471,9.948,149.562
C00680=1114.137,250.389,-71.779,-178.475,9.946,149.562
C00681=1114.142,250.141,-71.751,-178.478,9.942,149.562
C00682=1114.146,249.892,-71.723,-178.482,9.940,149.562
C00683=1114.150,249.643,-71.694,-178.485,9.936,149.562
C00684=1114.154,249.396,-71.665,-178.489,9.933,149.563
C00685=1114.159,249.147,-71.637,-178.493,9.930,149.563
C00686=1114.163,248.899,-71.609,-178.497,9.926,149.563
C00687=1114.167,248.651,-71.581,-178.501,9.923,149.563
C00688=1114.171,248.402,-71.552,-178.504,9.920,149.563
C00689=1114.176,248.154,-71.524,-178.508,9.916,149.564
C00690=1114.180,247.905,-71.495,-178.512,9.912,149.564
C00691=1114.185,247.657,-71.468,-178.516,9.909,149.564
C00692=1114.188,247.409,-71.440,-178.520,9.905,149.564
C00693=1114.193,247.161,-71.411,-178.521,9.903,149.564
C00694=1114.197,246.912,-71.383,-178.524,9.900,149.564
C00695=1114.201,246.664,-71.355,-178.526,9.897,149.564
C00696=1114.206,246.415,-71.327,-178.528,9.895,149.564
C00697=1114.210,246.167,-71.299,-178.531,9.892,149.564
C00698=1114.214,245.919,-71.271,-178.533,9.890,149.564
C00699=1114.219,245.671,-71.242,-178.535,9.887,149.564
C00700=1114.223,245.422,-71.214,-178.537,9.884,149.564
C00701=1114.227,245.174,-71.186,-178.539,9.882,149.564
C00702=1114.232,244.925,-71.158,-178.541,9.879,149.563
C00703=1114.236,244.677,-71.131,-178.544,9.877,149.564
C00704=1114.240,244.428,-71.102,-178.546,9.874,149.564
C00705=1114.244,244.180,-71.075,-178.548,9.871,149.563
C00706=1114.249,243.931,-71.046,-178.551,9.870,149.564
C00707=1114.253,243.684,-71.018,-178.553,9.866,149.564
C00708=1114.257,243.434,-70.991,-178.555,9.864,149.563
C00709=1114.262,243.186,-70.963,-178.558,9.861,149.564
C00710=1114.266,242.938,-70.934,-178.560,9.859,149.564
C00711=1114.271,242.690,-70.906,-178.563,9.856,149.564
C00712=1114.274,242.441,-70.878,-178.565,9.854,149.564
C00713=1114.279,242.193,-70.851,-178.568,9.851,149.564
C00714=1114.283,241.945,-70.823,-178.569,9.849,149.564
C00715=1114.288,241.696,-70.795,-178.572,9.846,149.564
C00716=1114.292,241.448,-70.767,-178.574,9.844,149.564
C00717=1114.296,241.199,-70.739,-178.577,9.841,149.564
C00718=1114.301,240.951,-70.712,-178.579,9.839,149.564
C00719=1114.304,240.702,-70.684,-178.582,9.836,149.564
C00720=1114.309,240.489,-70.659,-178.584,9.834,149.564
C00721=1114.313,240.276,-70.636,-178.586,9.832,149.564
C00722=1114.316,240.063,-70.612,-178.589,9.830,149.564
C00723=1114.320,239.850,-70.589,-178.591,9.827,149.564
C00724=1114.323,239.638,-70.565,-178.593,9.825,149.564
C00725=1114.327,239.425,-70.541,-178.595,9.823,149.564
C00726=1114.331,239.210,-70.517,-178.597,9.821,149.564
C00727=1114.335,238.997,-70.493,-178.599,9.819,149.564
C00728=1114.339,238.750,-70.465,-178.602,9.816,149.564
C00729=1114.343,238.500,-70.438,-178.605,9.813,149.564
C00730=1114.348,238.253,-70.410,-178.607,9.811,149.565
C00731=1114.352,238.004,-70.383,-178.610,9.808,149.565
C00732=1114.356,237.755,-70.355,-178.613,9.805,149.565
C00733=1114.361,237.507,-70.328,-178.615,9.803,149.565
C00734=1114.365,237.259,-70.300,-178.618,9.801,149.565
C00735=1114.369,237.010,-70.273,-178.621,9.798,149.565
C00736=1114.373,236.762,-70.245,-178.623,9.796,149.565
C00737=1114.378,236.514,-70.218,-178.626,9.793,149.565
C00738=1114.382,236.265,-70.190,-178.629,9.790,149.565
C00739=1114.386,236.016,-70.163,-178.632,9.787,149.565
C00740=1114.391,235.769,-70.135,-178.634,9.785,149.565
C00741=1114.395,235.519,-70.108,-178.637,9.783,149.566
C00742=1114.399,235.271,-70.080,-178.640,9.780,149.566
C00743=1114.404,235.023,-70.053,-178.642,9.777,149.566
C00744=1114.408,234.775,-70.026,-178.645,9.774,149.566
C00745=1114.412,234.526,-69.997,-178.648,9.771,149.566
C00746=1114.417,234.277,-69.970,-178.650,9.769,149.566
C00747=1114.422,234.029,-69.943,-178.653,9.766,149.566
C00748=1114.425,233.780,-69.915,-178.656,9.764,149.566
C00749=1114.430,233.532,-69.888,-178.659,9.761,149.566
C00750=1114.435,233.283,-69.861,-178.662,9.758,149.566
C00751=1114.439,233.035,-69.833,-178.665,9.755,149.566
C00752=1114.443,232.786,-69.806,-178.668,9.752,149.567
C00753=1114.448,232.538,-69.779,-178.671,9.750,149.567
C00754=1114.452,232.290,-69.752,-178.673,9.747,149.567
C00755=1114.456,232.042,-69.725,-178.676,9.744,149.567
C00756=1114.460,231.793,-69.697,-178.679,9.741,149.567
C00757=1114.465,231.544,-69.670,-178.682,9.738,149.567
C00758=1114.469,231.296,-69.643,-178.685,9.736,149.567
C00759=1114.474,231.047,-69.616,-178.688,9.732,149.567
C00760=1114.478,230.799,-69.588,-178.690,9.730,149.567
C00761=1114.482,230.550,-69.561,-178.694,9.726,149.567
C00762=1114.486,230.302,-69.534,-178.697,9.723,149.567
C00763=1114.491,230.053,-69.507,-178.700,9.720,149.567
C00764=1114.496,229.805,-69.480,-178.702,9.718,149.568
C00765=1114.500,229.556,-69.453,-178.705,9.715,149.568
C00766=1114.504,229.308,-69.427,-178.709,9.711,149.568
C00767=1114.508,229.059,-69.399,-178.711,9.708,149.568
C00768=1114.513,228.810,-69.372,-178.714,9.705,149.568
C00769=1114.518,228.562,-69.345,-178.717,9.702,149.568
C00770=1114.521,228.314,-69.319,-178.720,9.700,149.568
C00771=1114.526,228.065,-69.292,-178.723,9.696,149.568
C00772=1114.531,227.817,-69.265,-178.726,9.693,149.568
C00773=1114.534,227.568,-69.238,-178.729,9.690,149.568
C00774=1114.539,227.319,-69.211,-178.731,9.687,149.568
C00775=1114.543,227.071,-69.184,-178.734,9.684,149.568
C00776=1114.547,226.858,-69.160,-178.737,9.681,149.568
C00777=1114.550,226.645,-69.138,-178.738,9.678,149.568
C00778=1114.554,226.432,-69.114,-178.741,9.676,149.568
C00779=1114.558,226.218,-69.091,-178.743,9.673,149.568
C00780=1114.563,226.006,-69.068,-178.746,9.670,149.568
C00781=1114.566,225.793,-69.046,-178.748,9.668,149.568
C00782=1114.570,225.579,-69.023,-178.750,9.665,149.568
C00783=1114.573,225.366,-68.999,-178.753,9.662,149.568
C00784=1114.578,225.117,-68.973,-178.756,9.659,149.568
C00785=1114.582,224.869,-68.946,-178.758,9.656,149.568
C00786=1114.587,224.620,-68.919,-178.761,9.653,149.568
C00787=1114.591,224.372,-68.893,-178.763,9.650,149.568
C00788=1114.595,224.123,-68.865,-178.766,9.647,149.567
C00789=1114.600,223.874,-68.839,-178.768,9.643,149.567
C00790=1114.604,223.626,-68.813,-178.771,9.640,149.567
C00791=1114.608,223.377,-68.786,-178.774,9.638,149.567
C00792=1114.612,223.129,-68.759,-178.776,9.634,149.567
C00793=1114.617,222.880,-68.733,-178.779,9.631,149.567
C00794=1114.621,222.632,-68.706,-178.781,9.628,149.567
C00795=1114.626,222.383,-68.679,-178.784,9.625,149.567
C00796=1114.630,222.135,-68.653,-178.786,9.622,149.567
C00797=1114.635,221.886,-68.626,-178.789,9.619,149.567
C00798=1114.639,221.638,-68.600,-178.791,9.615,149.567
C00799=1114.644,221.389,-68.574,-178.794,9.612,149.567
C00800=1114.647,221.140,-68.547,-178.796,9.609,149.567
C00801=1114.652,220.892,-68.520,-178.799,9.606,149.567
C00802=1114.656,220.643,-68.494,-178.801,9.603,149.567
C00803=1114.661,220.395,-68.467,-178.804,9.600,149.566
C00804=1114.665,220.146,-68.441,-178.806,9.598,149.566
C00805=1114.670,219.897,-68.414,-178.808,9.594,149.566
C00806=1114.674,219.649,-68.388,-178.810,9.591,149.566
C00807=1114.678,219.400,-68.362,-178.813,9.588,149.566
C00808=1114.683,219.153,-68.336,-178.815,9.585,149.566
C00809=1114.688,218.904,-68.310,-178.818,9.582,149.566
C00810=1114.692,218.655,-68.283,-178.820,9.579,149.566
C00811=1114.696,218.406,-68.257,-178.822,9.576,149.566
C00812=1114.700,218.158,-68.231,-178.824,9.573,149.565
C00813=1114.705,217.909,-68.204,-178.827,9.570,149.565
C00814=1114.709,217.661,-68.178,-178.829,9.567,149.565
C00815=1114.713,217.412,-68.152,-178.831,9.563,149.565
C00816=1114.718,217.164,-68.125,-178.833,9.561,149.565
C00817=1114.722,216.915,-68.099,-178.836,9.558,149.565
C00818=1114.727,216.666,-68.073,-178.838,9.555,149.565
C00819=1114.731,216.418,-68.046,-178.840,9.552,149.565
C00820=1114.735,216.169,-68.021,-178.842,9.549,149.565
C00821=1114.740,215.921,-67.994,-178.845,9.546,149.565
C00822=1114.745,215.672,-67.968,-178.847,9.543,149.564
C00823=1114.749,215.423,-67.942,-178.849,9.540,149.564
C00824=1114.753,215.175,-67.916,-178.851,9.537,149.564
C00825=1114.758,214.926,-67.890,-178.853,9.534,149.564
C00826=1114.762,214.677,-67.864,-178.855,9.531,149.564
C00827=1114.766,214.429,-67.837,-178.858,9.528,149.564
C00828=1114.770,214.180,-67.812,-178.860,9.525,149.564
C00829=1114.776,213.932,-67.786,-178.862,9.522,149.564
C00830=1114.780,213.683,-67.760,-178.864,9.520,149.563
C00831=1114.784,213.435,-67.733,-178.866,9.516,149.563
C00832=1114.787,213.222,-67.711,-178.868,9.514,149.563
C00833=1114.791,213.008,-67.688,-178.871,9.511,149.563
C00834=1114.796,212.795,-67.667,-178.873,9.509,149.563
C00835=1114.800,212.581,-67.645,-178.876,9.506,149.563
C00836=1114.803,212.368,-67.622,-178.878,9.504,149.563
C00837=1114.807,212.155,-67.601,-178.880,9.501,149.563
C00838=1114.811,211.941,-67.578,-178.882,9.498,149.563
C00839=1114.814,211.728,-67.556,-178.885,9.495,149.563
C00840=1114.818,211.479,-67.530,-178.887,9.492,149.563
C00841=1114.824,211.231,-67.504,-178.890,9.489,149.563
C00842=1114.828,210.982,-67.478,-178.893,9.486,149.563
C00843=1114.832,210.733,-67.452,-178.895,9.483,149.563
C00844=1114.836,210.485,-67.426,-178.898,9.480,149.563
C00845=1114.841,210.237,-67.400,-178.901,9.478,149.563
C00846=1114.845,209.988,-67.375,-178.903,9.474,149.563
C00847=1114.850,209.739,-67.349,-178.906,9.472,149.563
C00848=1114.854,209.491,-67.323,-178.909,9.469,149.564
C00849=1114.859,209.242,-67.297,-178.912,9.466,149.564
C00850=1114.864,208.993,-67.271,-178.915,9.463,149.564
C00851=1114.868,208.744,-67.246,-178.917,9.460,149.564
C00852=1114.872,208.496,-67.220,-178.920,9.457,149.564
C00853=1114.877,208.248,-67.195,-178.923,9.454,149.564
C00854=1114.881,207.999,-67.169,-178.926,9.451,149.564
C00855=1114.885,207.750,-67.143,-178.929,9.449,149.564
C00856=1114.890,207.501,-67.117,-178.931,9.446,149.564
C00857=1114.894,207.253,-67.092,-178.934,9.443,149.564
C00858=1114.899,207.004,-67.067,-178.937,9.440,149.564
C00859=1114.903,206.755,-67.041,-178.940,9.437,149.564
C00860=1114.908,206.507,-67.016,-178.943,9.434,149.564
C00861=1114.912,206.258,-66.990,-178.946,9.431,149.564
C00862=1114.916,206.009,-66.964,-178.949,9.429,149.565
C00863=1114.921,205.761,-66.939,-178.951,9.426,149.565
C00864=1114.926,205.512,-66.913,-178.954,9.423,149.565
C00865=1114.930,205.263,-66.888,-178.958,9.419,149.565
C00866=1114.935,205.015,-66.863,-178.961,9.417,149.565
C00867=1114.939,204.766,-66.837,-178.963,9.413,149.565
C00868=1114.944,204.518,-66.812,-178.966,9.411,149.565
C00869=1114.948,204.269,-66.786,-178.969,9.408,149.565
C00870=1114.953,204.020,-66.761,-178.972,9.405,149.565
C00871=1114.957,203.772,-66.736,-178.974,9.402,149.565
C00872=1114.961,203.523,-66.710,-178.977,9.399,149.565
C00873=1114.966,203.274,-66.686,-178.980,9.397,149.566
C00874=1114.970,203.025,-66.660,-178.983,9.394,149.566
C00875=1114.975,202.777,-66.634,-178.986,9.391,149.566
C00876=1114.980,202.528,-66.609,-178.989,9.388,149.566
C00877=1114.984,202.279,-66.584,-178.992,9.385,149.566
C00878=1114.988,202.031,-66.559,-178.995,9.381,149.566
C00879=1114.993,201.782,-66.534,-178.998,9.379,149.566
C00880=1114.997,201.533,-66.508,-179.001,9.376,149.566
C00881=1115.002,201.285,-66.483,-179.003,9.373,149.566
C00882=1115.006,201.036,-66.458,-179.006,9.370,149.566
C00883=1115.010,200.788,-66.433,-179.009,9.367,149.566
C00884=1115.015,200.538,-66.408,-179.012,9.363,149.566
C00885=1115.020,200.290,-66.382,-179.015,9.361,149.566
C00886=1115.024,200.041,-66.357,-179.018,9.358,149.567
C00887=1115.028,199.793,-66.333,-179.021,9.355,149.567
C00888=1115.032,199.579,-66.311,-179.024,9.352,149.567
C00889=1115.036,199.366,-66.290,-179.026,9.349,149.567
C00890=1115.039,199.152,-66.268,-179.029,9.347,149.567
C00891=1115.044,198.939,-66.247,-179.031,9.344,149.567
C00892=1115.047,198.725,-66.225,-179.033,9.342,149.567
C00893=1115.051,198.512,-66.204,-179.036,9.339,149.567
C00894=1115.055,198.299,-66.182,-179.038,9.336,149.567
C00895=1115.059,198.085,-66.161,-179.041,9.333,149.567
C00896=1115.063,197.836,-66.136,-179.044,9.330,149.567
C00897=1115.068,197.588,-66.110,-179.047,9.327,149.567
C00898=1115.072,197.339,-66.086,-179.049,9.324,149.567
C00899=1115.077,197.090,-66.061,-179.053,9.320,149.567
C00900=1115.081,196.842,-66.036,-179.055,9.317,149.567
C00901=1115.086,196.593,-66.011,-179.059,9.314,149.567
C00902=1115.090,196.343,-65.986,-179.061,9.310,149.567
C00903=1115.095,196.095,-65.962,-179.063,9.308,149.567
C00904=1115.100,195.847,-65.937,-179.065,9.305,149.567
C00905=1115.104,195.597,-65.912,-179.067,9.302,149.567
C00906=1115.108,195.349,-65.888,-179.069,9.300,149.566
C00907=1115.113,195.100,-65.862,-179.071,9.296,149.566
C00908=1115.117,194.852,-65.838,-179.073,9.294,149.566
C00909=1115.122,194.602,-65.813,-179.074,9.291,149.566
C00910=1115.126,194.354,-65.789,-179.077,9.288,149.566
C00911=1115.131,194.105,-65.764,-179.079,9.286,149.566
C00912=1115.135,193.857,-65.739,-179.081,9.283,149.566
C00913=1115.140,193.608,-65.714,-179.083,9.280,149.566
C00914=1115.144,193.359,-65.689,-179.085,9.277,149.566
C00915=1115.149,193.110,-65.665,-179.087,9.275,149.566
C00916=1115.154,192.862,-65.641,-179.089,9.272,149.566
C00917=1115.158,192.612,-65.616,-179.091,9.269,149.565
C00918=1115.162,192.364,-65.591,-179.093,9.267,149.565
C00919=1115.167,192.116,-65.567,-179.096,9.264,149.565
C00920=1115.171,191.866,-65.542,-179.098,9.261,149.565
C00921=1115.176,191.618,-65.518,-179.100,9.258,149.565
C00922=1115.181,191.369,-65.493,-179.102,9.256,149.565
C00923=1115.185,191.120,-65.469,-179.104,9.253,149.565
C00924=1115.189,190.872,-65.444,-179.106,9.250,149.565
C00925=1115.194,190.623,-65.420,-179.108,9.247,149.565
C00926=1115.198,190.374,-65.395,-179.110,9.244,149.565
C00927=1115.203,190.125,-65.371,-179.113,9.241,149.565
C00928=1115.207,189.877,-65.347,-179.115,9.239,149.565
C00929=1115.212,189.627,-65.322,-179.117,9.236,149.565
C00930=1115.216,189.379,-65.297,-179.120,9.233,149.565
C00931=1115.221,189.131,-65.273,-179.122,9.230,149.565
C00932=1115.225,188.881,-65.248,-179.124,9.227,149.564
C00933=1115.230,188.633,-65.224,-179.126,9.225,149.564
C00934=1115.235,188.384,-65.200,-179.129,9.222,149.564
C00935=1115.239,188.135,-65.175,-179.131,9.219,149.564
C00936=1115.243,187.886,-65.151,-179.133,9.217,149.564
C00937=1115.248,187.638,-65.126,-179.136,9.213,149.564
C00938=1115.253,187.389,-65.102,-179.137,9.211,149.564
C00939=1115.256,187.140,-65.078,-179.140,9.208,149.564
C00940=1115.262,186.892,-65.053,-179.143,9.205,149.564
C00941=1115.266,186.642,-65.030,-179.145,9.202,149.564
C00942=1115.271,186.394,-65.006,-179.147,9.200,149.564
C00943=1115.275,186.145,-64.981,-179.150,9.197,149.564
C00944=1115.279,185.932,-64.960,-179.152,9.194,149.564
C00945=1115.283,185.718,-64.940,-179.154,9.192,149.564
C00946=1115.287,185.505,-64.919,-179.156,9.189,149.564
C00947=1115.290,185.291,-64.898,-179.158,9.187,149.564
C00948=1115.295,185.077,-64.877,-179.160,9.184,149.564
C00949=1115.299,184.864,-64.856,-179.162,9.182,149.564
C00950=1115.302,184.650,-64.835,-179.164,9.180,149.564
C00951=1115.306,184.436,-64.815,-179.166,9.176,149.564
C00952=1115.311,184.188,-64.791,-179.169,9.173,149.564
C00953=1115.315,183.939,-64.767,-179.171,9.171,149.564
C00954=1115.320,183.691,-64.742,-179.173,9.168,149.564
C00955=1115.324,183.441,-64.719,-179.176,9.165,149.564
C00956=1115.329,183.193,-64.694,-179.179,9.162,149.564
C00957=1115.333,182.944,-64.670,-179.181,9.159,149.564
C00958=1115.338,182.695,-64.647,-179.184,9.156,149.564
C00959=1115.343,182.446,-64.622,-179.186,9.153,149.564
C00960=1115.347,182.198,-64.598,-179.189,9.150,149.564
C00961=1115.351,181.948,-64.575,-179.191,9.147,149.564
C00962=1115.356,181.700,-64.551,-179.193,9.144,149.564
C00963=1115.361,181.451,-64.527,-179.196,9.141,149.564
C00964=1115.365,181.202,-64.503,-179.198,9.138,149.564
C00965=1115.369,180.954,-64.479,-179.201,9.135,149.564
C00966=1115.375,180.705,-64.455,-179.203,9.132,149.563
C00967=1115.379,180.456,-64.431,-179.206,9.129,149.563
C00968=1115.383,180.207,-64.407,-179.208,9.126,149.563
C00969=1115.388,179.958,-64.383,-179.212,9.122,149.563
C00970=1115.392,179.709,-64.360,-179.214,9.119,149.563
C00971=1115.397,179.461,-64.336,-179.217,9.115,149.563
C00972=1115.401,179.212,-64.312,-179.219,9.112,149.563
C00973=1115.406,178.963,-64.288,-179.221,9.110,149.563
C00974=1115.411,178.714,-64.265,-179.223,9.107,149.563
C00975=1115.415,178.466,-64.241,-179.225,9.104,149.563
C00976=1115.419,178.216,-64.217,-179.227,9.101,149.563
C00977=1115.423,177.968,-64.193,-179.230,9.098,149.563
C00978=1115.428,177.719,-64.170,-179.231,9.095,149.563
C00979=1115.433,177.470,-64.146,-179.234,9.092,149.562
C00980=1115.437,177.221,-64.122,-179.236,9.089,149.562
C00981=1115.442,176.972,-64.099,-179.238,9.086,149.562
C00982=1115.446,176.724,-64.075,-179.240,9.083,149.562
C00983=1115.451,176.475,-64.051,-179.243,9.080,149.562
C00984=1115.456,176.226,-64.028,-179.244,9.077,149.562
C00985=1115.460,175.977,-64.004,-179.247,9.074,149.562
C00986=1115.465,175.728,-63.981,-179.249,9.071,149.562
C00987=1115.469,175.479,-63.957,-179.251,9.068,149.562
C00988=1115.474,175.230,-63.934,-179.254,9.065,149.562
C00989=1115.479,174.982,-63.910,-179.256,9.062,149.561
C00990=1115.483,174.733,-63.887,-179.258,9.060,149.561
C00991=1115.488,174.484,-63.863,-179.260,9.056,149.561
C00992=1115.492,174.235,-63.839,-179.262,9.053,149.561
C00993=1115.497,173.986,-63.816,-179.264,9.051,149.561
C00994=1115.502,173.737,-63.792,-179.267,9.048,149.561
C00995=1115.506,173.488,-63.770,-179.269,9.044,149.561
C00996=1115.510,173.239,-63.746,-179.271,9.042,149.561
C00997=1115.515,172.991,-63.722,-179.273,9.039,149.561
C00998=1115.520,172.742,-63.699,-179.275,9.035,149.560
C00999=1115.524,172.493,-63.675,-179.277,9.033,149.560
C01000=1115.528,172.279,-63.656,-179.280,9.030,149.560
C01001=1115.533,172.066,-63.635,-179.281,9.027,149.560
C01002=1115.536,171.852,-63.615,-179.283,9.025,149.560
C01003=1115.540,171.638,-63.596,-179.285,9.022,149.560
C01004=1115.544,171.425,-63.576,-179.287,9.020,149.560
C01005=1115.548,171.211,-63.555,-179.288,9.017,149.560
C01006=1115.552,170.997,-63.535,-179.291,9.014,149.560
C01007=1115.555,170.783,-63.515,-179.293,9.012,149.560
C01008=1115.560,170.535,-63.492,-179.295,9.009,149.560
C01009=1115.565,170.286,-63.468,-179.297,9.006,149.559
C01010=1115.570,170.037,-63.445,-179.299,9.003,149.559
C01011=1115.574,169.789,-63.422,-179.302,9.000,149.559
C01012=1115.578,169.540,-63.399,-179.304,8.996,149.559
C01013=1115.583,169.291,-63.376,-179.306,8.994,149.559
C01014=1115.588,169.042,-63.352,-179.308,8.991,149.559
C01015=1115.592,168.793,-63.329,-179.310,8.987,149.559
C01016=1115.596,168.544,-63.306,-179.312,8.985,149.559
C01017=1115.601,168.295,-63.283,-179.315,8.982,149.559
C01018=1115.606,168.046,-63.260,-179.317,8.978,149.558
C01019=1115.610,167.798,-63.237,-179.319,8.975,149.558
C01020=1115.615,167.548,-63.214,-179.322,8.972,149.558
C01021=1115.620,167.299,-63.191,-179.323,8.970,149.558
C01022=1115.624,167.050,-63.168,-179.326,8.966,149.558
C01023=1115.629,166.801,-63.145,-179.328,8.963,149.558
C01024=1115.633,166.552,-63.122,-179.330,8.960,149.558
C01025=1115.639,166.304,-63.099,-179.332,8.957,149.558
C01026=1115.643,166.055,-63.076,-179.335,8.954,149.558
C01027=1115.647,165.806,-63.052,-179.337,8.951,149.558
C01028=1115.652,165.557,-63.030,-179.339,8.948,149.558
C01029=1115.656,165.308,-63.007,-179.341,8.944,149.557
C01030=1115.662,165.059,-62.984,-179.343,8.942,149.557
C01031=1115.666,164.811,-62.961,-179.346,8.939,149.557
C01032=1115.670,164.562,-62.938,-179.348,8.935,149.557
C01033=1115.675,164.313,-62.915,-179.350,8.932,149.557
C01034=1115.679,164.063,-62.892,-179.353,8.929,149.557
C01035=1115.684,163.814,-62.869,-179.355,8.926,149.557
C01036=1115.689,163.566,-62.847,-179.357,8.923,149.557
C01037=1115.694,163.317,-62.824,-179.359,8.920,149.556
C01038=1115.698,163.068,-62.801,-179.362,8.917,149.556
C01039=1115.702,162.819,-62.778,-179.364,8.913,149.556
C01040=1115.708,162.571,-62.755,-179.366,8.910,149.556
C01041=1115.712,162.321,-62.733,-179.369,8.907,149.556
C01042=1115.717,162.072,-62.710,-179.370,8.904,149.556
C01043=1115.720,161.823,-62.687,-179.373,8.901,149.556
C01044=1115.726,161.574,-62.665,-179.375,8.898,149.556
C01045=1115.730,161.326,-62.642,-179.377,8.895,149.555
C01046=1115.735,161.077,-62.618,-179.379,8.891,149.555
C01047=1115.739,160.827,-62.596,-179.382,8.888,149.555
C01048=1115.744,160.579,-62.573,-179.384,8.885,149.555
C01049=1115.749,160.330,-62.551,-179.386,8.881,149.555
C01050=1115.753,160.081,-62.529,-179.389,8.878,149.555
C01051=1115.758,159.831,-62.506,-179.390,8.876,149.555
C01052=1115.762,159.583,-62.483,-179.393,8.872,149.554
C01053=1115.767,159.334,-62.460,-179.395,8.869,149.554
C01054=1115.771,159.085,-62.438,-179.397,8.866,149.554
C01055=1115.776,158.837,-62.415,-179.400,8.862,149.554
C01056=1115.780,158.622,-62.396,-179.402,8.859,149.554
C01057=1115.784,158.409,-62.377,-179.404,8.857,149.554
C01058=1115.788,158.195,-62.358,-179.406,8.854,149.554
C01059=1115.792,157.981,-62.339,-179.408,8.851,149.554
C01060=1115.795,157.767,-62.319,-179.409,8.848,149.554
C01061=1115.800,157.553,-62.300,-179.412,8.845,149.553
C01062=1115.804,157.340,-62.280,-179.413,8.843,149.553
C01063=1115.808,157.126,-62.261,-179.415,8.840,149.553
C01064=1115.812,156.877,-62.238,-179.417,8.837,149.553
C01065=1115.818,156.628,-62.216,-179.420,8.833,149.553
C01066=1115.822,156.379,-62.194,-179.422,8.830,149.553
C01067=1115.826,156.130,-62.171,-179.424,8.827,149.553
C01068=1115.831,155.881,-62.149,-179.426,8.823,149.552
C01069=1115.836,155.632,-62.127,-179.428,8.820,149.552
C01070=1115.840,155.383,-62.104,-179.431,8.817,149.552
C01071=1115.845,155.134,-62.082,-179.433,8.813,149.552
C01072=1115.850,154.885,-62.060,-179.435,8.810,149.552
C01073=1115.854,154.637,-62.038,-179.437,8.807,149.552
C01074=1115.858,154.388,-62.015,-179.440,8.803,149.551
C01075=1115.863,154.138,-61.993,-179.442,8.800,149.551
C01076=1115.868,153.890,-61.970,-179.444,8.796,149.551
C01077=1115.872,153.641,-61.948,-179.447,8.792,149.551
C01078=1115.877,153.392,-61.927,-179.449,8.789,149.551
C01079=1115.882,153.142,-61.904,-179.451,8.786,149.551
C01080=1115.887,152.894,-61.882,-179.454,8.782,149.550
C01081=1115.891,152.645,-61.860,-179.456,8.779,149.550
C01082=1115.896,152.396,-61.838,-179.458,8.775,149.550
C01083=1115.901,152.147,-61.815,-179.460,8.772,149.550
C01084=1115.905,151.897,-61.793,-179.462,8.769,149.550
C01085=1115.910,151.649,-61.772,-179.464,8.765,149.549
C01086=1115.914,151.399,-61.750,-179.467,8.762,149.549
C01087=1115.919,151.151,-61.727,-179.469,8.758,149.549
C01088=1115.923,150.902,-61.705,-179.472,8.754,149.549
C01089=1115.929,150.653,-61.683,-179.474,8.751,149.549
C01090=1115.933,150.404,-61.661,-179.476,8.747,149.548
C01091=1115.938,150.155,-61.639,-179.478,8.744,149.548
C01092=1115.942,149.906,-61.617,-179.480,8.740,149.548
C01093=1115.947,149.657,-61.595,-179.482,8.737,149.548
C01094=1115.951,149.408,-61.573,-179.484,8.733,149.547
C01095=1115.956,149.159,-61.552,-179.487,8.729,149.547
C01096=1115.961,148.910,-61.530,-179.489,8.726,149.547
C01097=1115.966,148.661,-61.507,-179.492,8.722,149.547
C01098=1115.971,148.412,-61.486,-179.494,8.719,149.547
C01099=1115.975,148.163,-61.464,-179.496,8.715,149.546
C01100=1115.980,147.914,-61.442,-179.498,8.711,149.546
C01101=1115.984,147.665,-61.420,-179.500,8.708,149.546
C01102=1115.989,147.416,-61.398,-179.503,8.704,149.546
C01103=1115.993,147.167,-61.376,-179.505,8.701,149.545
C01104=1115.998,146.918,-61.354,-179.507,8.696,149.545
C01105=1116.003,146.669,-61.333,-179.509,8.693,149.545
C01106=1116.008,146.420,-61.311,-179.512,8.689,149.545
C01107=1116.012,146.171,-61.290,-179.514,8.686,149.545
C01108=1116.017,145.922,-61.268,-179.516,8.682,149.544
C01109=1116.022,145.673,-61.246,-179.518,8.678,149.544
C01110=1116.026,145.424,-61.224,-179.520,8.674,149.544
C01111=1116.031,145.174,-61.203,-179.522,8.671,149.543
C01112=1116.035,144.961,-61.185,-179.524,8.667,149.543
C01113=1116.039,144.747,-61.166,-179.526,8.665,149.543
C01114=1116.042,144.533,-61.147,-179.527,8.662,149.542
C01115=1116.047,144.320,-61.129,-179.528,8.659,149.542
C01116=1116.050,144.106,-61.110,-179.530,8.656,149.542
C01117=1116.055,143.892,-61.091,-179.531,8.653,149.542
C01118=1116.059,143.678,-61.074,-179.532,8.650,149.541
C01119=1116.063,143.464,-61.054,-179.533,8.648,149.541
C01120=1116.068,143.215,-61.033,-179.535,8.644,149.541
C01121=1116.072,142.966,-61.011,-179.537,8.640,149.540
C01122=1116.077,142.716,-60.990,-179.538,8.637,149.540
C01123=1116.081,142.468,-60.969,-179.540,8.634,149.540
C01124=1116.086,142.219,-60.947,-179.541,8.631,149.539
C01125=1116.091,141.970,-60.926,-179.543,8.627,149.539
C01126=1116.096,141.721,-60.904,-179.545,8.623,149.539
C01127=1116.100,141.472,-60.882,-179.546,8.621,149.538
C01128=1116.105,141.222,-60.861,-179.548,8.617,149.538
C01129=1116.110,140.974,-60.839,-179.550,8.613,149.538
C01130=1116.113,140.725,-60.818,-179.551,8.610,149.537
C01131=1116.119,140.475,-60.797,-179.553,8.607,149.537
C01132=1116.124,140.227,-60.775,-179.555,8.603,149.537
C01133=1116.129,139.977,-60.754,-179.556,8.600,149.536
C01134=1116.133,139.728,-60.732,-179.558,8.597,149.536
C01135=1116.137,139.479,-60.712,-179.559,8.593,149.536
C01136=1116.142,139.231,-60.690,-179.561,8.590,149.536
C01137=1116.147,138.981,-60.668,-179.563,8.586,149.535
C01138=1116.152,138.732,-60.647,-179.565,8.583,149.535
C01139=1116.156,138.484,-60.626,-179.567,8.580,149.535
C01140=1116.161,138.234,-60.605,-179.568,8.576,149.534
C01141=1116.165,137.985,-60.583,-179.570,8.573,149.534
C01142=1116.170,137.736,-60.562,-179.571,8.569,149.534
C01143=1116.175,137.487,-60.541,-179.573,8.567,149.533
C01144=1116.180,137.238,-60.520,-179.575,8.563,149.533
C01145=1116.184,136.989,-60.498,-179.576,8.559,149.533
C01146=1116.188,136.740,-60.478,-179.578,8.557,149.532
C01147=1116.194,136.491,-60.457,-179.580,8.553,149.532
C01148=1116.199,136.242,-60.435,-179.582,8.549,149.532
C01149=1116.204,135.993,-60.414,-179.583,8.547,149.532
C01150=1116.207,135.744,-60.392,-179.585,8.543,149.531
C01151=1116.212,135.494,-60.372,-179.586,8.540,149.531
C01152=1116.218,135.245,-60.351,-179.588,8.537,149.531
C01153=1116.222,134.997,-60.329,-179.590,8.533,149.530
C01154=1116.227,134.748,-60.308,-179.591,8.530,149.530
C01155=1116.231,134.498,-60.287,-179.593,8.526,149.530
C01156=1116.236,134.249,-60.266,-179.595,8.523,149.530
C01157=1116.241,134.000,-60.245,-179.596,8.520,149.529
C01158=1116.245,133.751,-60.225,-179.599,8.516,149.529
C01159=1116.250,133.502,-60.203,-179.601,8.513,149.529
C01160=1116.255,133.252,-60.182,-179.602,8.510,149.528
C01161=1116.259,133.003,-60.161,-179.604,8.506,149.528
C01162=1116.264,132.755,-60.140,-179.606,8.503,149.528
C01163=1116.268,132.506,-60.119,-179.607,8.500,149.527
C01164=1116.274,132.257,-60.098,-179.609,8.496,149.527
C01165=1116.279,132.007,-60.077,-179.610,8.493,149.527
C01166=1116.283,131.759,-60.056,-179.612,8.490,149.527
C01167=1116.287,131.509,-60.035,-179.614,8.486,149.526
C01168=1116.292,131.295,-60.018,-179.615,8.483,149.526
C01169=1116.296,131.082,-60.000,-179.617,8.481,149.526
C01170=1116.299,130.868,-59.982,-179.618,8.478,149.526
C01171=1116.304,130.654,-59.964,-179.620,8.475,149.525
C01172=1116.308,130.439,-59.946,-179.621,8.473,149.525
C01173=1116.312,130.226,-59.928,-179.623,8.469,149.525
C01174=1116.316,130.011,-59.910,-179.625,8.466,149.525
C01175=1116.320,129.798,-59.893,-179.626,8.464,149.524
C01176=1116.325,129.548,-59.872,-179.628,8.460,149.524
C01177=1116.329,129.299,-59.851,-179.629,8.457,149.524
C01178=1116.334,129.051,-59.830,-179.631,8.454,149.523
C01179=1116.339,128.802,-59.809,-179.633,8.450,149.523
C01180=1116.344,128.553,-59.788,-179.634,8.447,149.523
C01181=1116.348,128.304,-59.768,-179.636,8.443,149.523
C01182=1116.353,128.054,-59.746,-179.638,8.440,149.522
C01183=1116.357,127.805,-59.726,-179.639,8.437,149.522
C01184=1116.362,127.555,-59.705,-179.642,8.433,149.522
C01185=1116.367,127.306,-59.685,-179.644,8.430,149.521
C01186=1116.372,127.057,-59.664,-179.645,8.427,149.521
C01187=1116.377,126.808,-59.643,-179.647,8.423,149.521
C01188=1116.381,126.559,-59.623,-179.649,8.420,149.521
C01189=1116.386,126.310,-59.602,-179.650,8.417,149.520
C01190=1116.391,126.061,-59.582,-179.652,8.414,149.520
C01191=1116.396,125.812,-59.561,-179.654,8.410,149.520
C01192=1116.400,125.563,-59.540,-179.655,8.407,149.519
C01193=1116.405,125.314,-59.520,-179.657,8.403,149.519
C01194=1116.410,125.065,-59.499,-179.659,8.400,149.519
C01195=1116.414,124.816,-59.479,-179.661,8.397,149.519
C01196=1116.419,124.567,-59.458,-179.663,8.393,149.518
C01197=1116.424,124.318,-59.437,-179.665,8.390,149.518
C01198=1116.429,124.068,-59.418,-179.667,8.386,149.518
C01199=1116.433,123.819,-59.397,-179.668,8.384,149.518
C01200=1116.438,123.570,-59.376,-179.670,8.380,149.517
C01201=1116.443,123.321,-59.356,-179.672,8.376,149.517
C01202=1116.447,123.072,-59.336,-179.673,8.374,149.517
C01203=1116.452,122.823,-59.315,-179.675,8.370,149.517
C01204=1116.457,122.574,-59.294,-179.677,8.366,149.516
C01205=1116.461,122.324,-59.275,-179.678,8.364,149.516
C01206=1116.466,122.075,-59.254,-179.680,8.360,149.516
C01207=1116.471,121.826,-59.233,-179.682,8.357,149.515
C01208=1116.476,121.577,-59.213,-179.685,8.353,149.515
C01209=1116.480,121.327,-59.193,-179.686,8.350,149.515
C01210=1116.485,121.078,-59.173,-179.688,8.346,149.515
C01211=1116.490,120.830,-59.152,-179.690,8.343,149.514
C01212=1116.495,120.581,-59.132,-179.692,8.339,149.514
C01213=1116.500,120.331,-59.112,-179.693,8.336,149.514
C01214=1116.504,120.082,-59.092,-179.695,8.333,149.513
C01215=1116.509,119.833,-59.071,-179.697,8.329,149.513
C01216=1116.514,119.584,-59.051,-179.698,8.327,149.513
C01217=1116.518,119.335,-59.031,-179.700,8.323,149.513
C01218=1116.523,119.086,-59.010,-179.702,8.319,149.512
C01219=1116.527,118.837,-58.990,-179.704,8.316,149.512
C01220=1116.532,118.587,-58.970,-179.705,8.313,149.512
C01221=1116.538,118.339,-58.950,-179.707,8.309,149.511
C01222=1116.543,118.089,-58.930,-179.709,8.306,149.511
C01223=1116.547,117.840,-58.910,-179.711,8.302,149.511
C01224=1116.551,117.626,-58.892,-179.713,8.299,149.511
C01225=1116.555,117.412,-58.875,-179.714,8.297,149.511
C01226=1116.559,117.197,-58.858,-179.716,8.294,149.510
C01227=1116.563,116.984,-58.841,-179.718,8.290,149.510
C01228=1116.567,116.770,-58.824,-179.719,8.288,149.510
C01229=1116.571,116.556,-58.806,-179.720,8.285,149.510
C01230=1116.575,116.341,-58.789,-179.721,8.282,149.509
C01231=1116.580,116.127,-58.772,-179.724,8.278,149.509
C01232=1116.584,115.878,-58.751,-179.725,8.276,149.509
C01233=1116.589,115.629,-58.732,-179.727,8.272,149.509
C01234=1116.593,115.380,-58.711,-179.729,8.269,149.508
C01235=1116.599,115.131,-58.692,-179.731,8.265,149.508
C01236=1116.603,114.882,-58.672,-179.733,8.261,149.508
C01237=1116.608,114.633,-58.652,-179.734,8.259,149.507
C01238=1116.612,114.384,-58.632,-179.736,8.255,149.507
C01239=1116.617,114.134,-58.612,-179.738,8.251,149.507
C01240=1116.622,113.885,-58.593,-179.740,8.248,149.507
C01241=1116.628,113.636,-58.572,-179.742,8.244,149.506
C01242=1116.632,113.386,-58.552,-179.743,8.241,149.506
C01243=1116.637,113.137,-58.532,-179.745,8.238,149.506
C01244=1116.641,112.888,-58.512,-179.747,8.234,149.505
C01245=1116.647,112.639,-58.493,-179.749,8.230,149.505
C01246=1116.651,112.390,-58.472,-179.751,8.227,149.505
C01247=1116.656,112.140,-58.453,-179.752,8.224,149.505
C01248=1116.660,111.891,-58.434,-179.754,8.221,149.504
C01249=1116.665,111.643,-58.414,-179.756,8.217,149.504
C01250=1116.670,111.393,-58.394,-179.758,8.213,149.504
C01251=1116.675,111.144,-58.374,-179.760,8.210,149.503
C01252=1116.680,110.896,-58.354,-179.762,8.206,149.503
C01253=1116.684,110.646,-58.335,-179.764,8.202,149.503
C01254=1116.689,110.396,-58.315,-179.766,8.199,149.503
C01255=1116.694,110.147,-58.295,-179.768,8.195,149.502
C01256=1116.699,109.899,-58.275,-179.770,8.191,149.502
C01257=1116.704,109.649,-58.256,-179.773,8.188,149.502
C01258=1116.708,109.399,-58.236,-179.775,8.184,149.502
C01259=1116.714,109.151,-58.217,-179.777,8.180,149.501
C01260=1116.718,108.902,-58.196,-179.779,8.176,149.501
C01261=1116.722,108.652,-58.177,-179.781,8.172,149.501
C01262=1116.727,108.404,-58.158,-179.783,8.169,149.501
C01263=1116.732,108.154,-58.138,-179.785,8.165,149.500
C01264=1116.737,107.904,-58.119,-179.787,8.161,149.500
C01265=1116.742,107.656,-58.100,-179.789,8.157,149.500
C01266=1116.747,107.406,-58.080,-179.791,8.154,149.499
C01267=1116.751,107.157,-58.060,-179.793,8.150,149.499
C01268=1116.756,106.908,-58.041,-179.795,8.146,149.499
C01269=1116.761,106.659,-58.021,-179.798,8.142,149.499
C01270=1116.766,106.409,-58.002,-179.800,8.138,149.498
C01271=1116.770,106.161,-57.983,-179.801,8.135,149.498
C01272=1116.775,105.911,-57.963,-179.803,8.131,149.498
C01273=1116.780,105.662,-57.944,-179.805,8.127,149.497
C01274=1116.785,105.413,-57.924,-179.808,8.123,149.497
C01275=1116.789,105.163,-57.905,-179.810,8.119,149.497
C01276=1116.794,104.915,-57.886,-179.811,8.116,149.496
C01277=1116.799,104.665,-57.866,-179.813,8.112,149.496
C01278=1116.804,104.416,-57.847,-179.815,8.108,149.496
C01279=1116.808,104.167,-57.828,-179.817,8.105,149.496
C01280=1116.813,103.953,-57.811,-179.819,8.101,149.495
C01281=1116.817,103.738,-57.795,-179.820,8.098,149.495
C01282=1116.821,103.524,-57.778,-179.822,8.095,149.495
C01283=1116.825,103.311,-57.762,-179.824,8.091,149.494
C01284=1116.829,103.096,-57.745,-179.825,8.088,149.494
C01285=1116.833,102.882,-57.729,-179.827,8.084,149.494
C01286=1116.838,102.668,-57.712,-179.828,8.081,149.493
C01287=1116.842,102.454,-57.696,-179.830,8.078,149.493
C01288=1116.846,102.204,-57.676,-179.832,8.074,149.493
C01289=1116.852,101.955,-57.657,-179.834,8.070,149.492
C01290=1116.856,101.706,-57.638,-179.836,8.067,149.492
C01291=1116.861,101.456,-57.619,-179.837,8.063,149.492
C01292=1116.865,101.207,-57.600,-179.839,8.059,149.491
C01293=1116.871,100.958,-57.581,-179.841,8.055,149.491
C01294=1116.875,100.709,-57.561,-179.843,8.051,149.491
C01295=1116.880,100.460,-57.543,-179.844,8.048,149.490
C01296=1116.885,100.210,-57.524,-179.847,8.043,149.490
C01297=1116.890,99.961,-57.505,-179.848,8.039,149.489
C01298=1116.894,99.712,-57.485,-179.850,8.035,149.489
C01299=1116.899,99.463,-57.467,-179.852,8.032,149.489
C01300=1116.904,99.213,-57.448,-179.854,8.028,149.488
C01301=1116.909,98.964,-57.428,-179.855,8.024,149.488
C01302=1116.913,98.715,-57.409,-179.857,8.020,149.487
C01303=1116.919,98.465,-57.391,-179.858,8.016,149.487
C01304=1116.923,98.216,-57.372,-179.860,8.013,149.487
C01305=1116.928,97.967,-57.352,-179.862,8.009,149.486
C01306=1116.933,97.718,-57.334,-179.864,8.005,149.486
C01307=1116.938,97.469,-57.315,-179.865,8.001,149.486
C01308=1116.943,97.220,-57.296,-179.867,7.997,149.485
C01309=1116.948,96.970,-57.277,-179.869,7.993,149.485
C01310=1116.952,96.721,-57.258,-179.870,7.990,149.484
C01311=1116.957,96.471,-57.240,-179.872,7.986,149.484
C01312=1116.962,96.223,-57.221,-179.873,7.982,149.483
C01313=1116.967,95.974,-57.202,-179.875,7.978,149.483
C01314=1116.972,95.724,-57.183,-179.877,7.974,149.482
C01315=1116.976,95.475,-57.165,-179.878,7.970,149.482
C01316=1116.981,95.225,-57.146,-179.880,7.966,149.482
C01317=1116.986,94.976,-57.127,-179.881,7.962,149.481
C01318=1116.991,94.727,-57.109,-179.883,7.958,149.481
C01319=1116.996,94.478,-57.089,-179.885,7.955,149.480
C01320=1117.001,94.229,-57.071,-179.886,7.951,149.480
C01321=1117.006,93.980,-57.052,-179.887,7.948,149.479
C01322=1117.010,93.730,-57.034,-179.889,7.944,149.479
C01323=1117.015,93.481,-57.015,-179.890,7.940,149.479
C01324=1117.020,93.231,-56.996,-179.892,7.936,149.478
C01325=1117.024,92.983,-56.977,-179.893,7.932,149.478
C01326=1117.029,92.733,-56.959,-179.895,7.928,149.477
C01327=1117.034,92.483,-56.940,-179.897,7.924,149.477
C01328=1117.039,92.235,-56.922,-179.898,7.920,149.476
C01329=1117.044,91.985,-56.904,-179.899,7.916,149.476
C01330=1117.050,91.736,-56.885,-179.901,7.912,149.475
C01331=1117.054,91.487,-56.866,-179.902,7.909,149.475
C01332=1117.058,91.237,-56.848,-179.904,7.905,149.475
C01333=1117.064,90.989,-56.829,-179.905,7.901,149.474
C01334=1117.068,90.739,-56.810,-179.907,7.897,149.474
C01335=1117.073,90.490,-56.792,-179.908,7.893,149.473
C01336=1117.078,90.235,-56.774,-179.909,7.889,149.473
C01337=1117.083,89.979,-56.755,-179.911,7.885,149.472
C01338=1117.088,89.725,-56.736,-179.913,7.881,149.472
C01339=1117.093,89.471,-56.717,-179.913,7.878,149.471
C01340=1117.098,89.221,-56.698,-179.915,7.874,149.471
C01341=1117.102,88.972,-56.680,-179.916,7.870,149.470
C01342=1117.107,88.722,-56.662,-179.918,7.866,149.470
C01343=1117.112,88.474,-56.643,-179.919,7.862,149.469
C01344=1117.117,88.224,-56.624,-179.920,7.859,149.469
C01345=1117.122,87.975,-56.606,-179.922,7.855,149.468
C01346=1117.127,87.725,-56.588,-179.923,7.851,149.468
C01347=1117.132,87.476,-56.570,-179.924,7.847,149.467
C01348=1117.136,87.227,-56.551,-179.925,7.844,149.467
C01349=1117.141,86.977,-56.533,-179.927,7.839,149.466
C01350=1117.146,86.728,-56.515,-179.928,7.836,149.466
C01351=1117.151,86.479,-56.497,-179.930,7.832,149.465
C01352=1117.155,86.267,-56.481,-179.931,7.829,149.465
C01353=1117.159,86.056,-56.466,-179.932,7.825,149.464
C01354=1117.163,85.844,-56.450,-179.933,7.822,149.464
C01355=1117.168,85.633,-56.435,-179.934,7.819,149.464
C01356=1117.172,85.421,-56.420,-179.935,7.816,149.463
C01357=1117.175,85.210,-56.403,-179.935,7.813,149.463
C01358=1117.179,84.998,-56.388,-179.937,7.809,149.462
C01359=1117.184,84.787,-56.373,-179.938,7.806,149.462
C01360=1117.189,84.538,-56.355,-179.939,7.802,149.461
C01361=1117.193,84.288,-56.337,-179.940,7.799,149.461
C01362=1117.198,84.039,-56.319,-179.941,7.794,149.460
C01363=1117.203,83.790,-56.301,-179.942,7.791,149.460
C01364=1117.208,83.541,-56.283,-179.944,7.787,149.459
C01365=1117.214,83.291,-56.264,-179.945,7.783,149.459
C01366=1117.218,83.042,-56.246,-179.946,7.780,149.458
C01367=1117.223,82.792,-56.228,-179.947,7.776,149.457
C01368=1117.228,82.543,-56.210,-179.949,7.772,149.457
C01369=1117.233,82.294,-56.192,-179.949,7.768,149.456
C01370=1117.238,82.045,-56.174,-179.951,7.764,149.456
C01371=1117.242,81.795,-56.156,-179.951,7.761,149.455
C01372=1117.247,81.546,-56.138,-179.953,7.757,149.455
C01373=1117.252,81.297,-56.120,-179.953,7.753,149.454
C01374=1117.257,81.047,-56.101,-179.955,7.750,149.454
C01375=1117.261,80.798,-56.084,-179.956,7.745,149.453
C01376=1117.266,80.549,-56.066,-179.957,7.742,149.453
C01377=1117.272,80.299,-56.048,-179.958,7.738,149.452
C01378=1117.277,80.050,-56.030,-179.959,7.735,149.452
C01379=1117.281,79.801,-56.012,-179.960,7.730,149.451
C01380=1117.286,79.552,-55.994,-179.961,7.727,149.451
C01381=1117.291,79.302,-55.976,-179.962,7.723,149.450
C01382=1117.296,79.053,-55.958,-179.963,7.720,149.450
C01383=1117.301,78.804,-55.940,-179.964,7.716,149.449
C01384=1117.305,78.554,-55.922,-179.965,7.713,149.448
C01385=1117.311,78.304,-55.905,-179.967,7.708,149.448
C01386=1117.316,78.055,-55.887,-179.967,7.705,149.447
C01387=1117.320,77.806,-55.869,-179.969,7.701,149.447
C01388=1117.325,77.557,-55.851,-179.969,7.697,149.446
C01389=1117.330,77.308,-55.833,-179.971,7.693,149.446
C01390=1117.335,77.058,-55.816,-179.971,7.690,149.445
C01391=1117.340,76.809,-55.798,-179.972,7.686,149.444
C01392=1117.344,76.594,-55.783,-179.974,7.683,149.444
C01393=1117.348,76.380,-55.768,-179.975,7.680,149.444
C01394=1117.352,76.166,-55.752,-179.976,7.676,149.443
C01395=1117.356,75.951,-55.736,-179.977,7.673,149.443
C01396=1117.360,75.738,-55.722,-179.978,7.670,149.442
C01397=1117.365,75.523,-55.707,-179.980,7.666,149.442
C01398=1117.369,75.308,-55.691,-179.981,7.663,149.442
C01399=1117.373,75.094,-55.676,-179.982,7.659,149.441
C01400=1117.378,74.845,-55.658,-179.983,7.656,149.441
C01401=1117.384,74.595,-55.641,-179.984,7.651,149.440
C01402=1117.388,74.346,-55.623,-179.986,7.647,149.440
C01403=1117.393,74.097,-55.606,-179.988,7.644,149.439
C01404=1117.398,73.847,-55.588,-179.989,7.640,149.439
C01405=1117.403,73.598,-55.570,-179.990,7.635,149.438
C01406=1117.408,73.349,-55.552,-179.992,7.631,149.438
C01407=1117.412,73.100,-55.536,-179.993,7.628,149.437
C01408=1117.417,72.850,-55.518,-179.995,7.624,149.437
C01409=1117.422,72.601,-55.500,-179.996,7.619,149.436
C01410=1117.427,72.351,-55.482,-179.998,7.615,149.436
C01411=1117.432,72.102,-55.464,-179.999,7.612,149.435
C01412=1117.437,71.853,-55.448,180.000,7.607,149.435
C01413=1117.441,71.604,-55.430,179.998,7.603,149.434
C01414=1117.447,71.354,-55.412,179.997,7.600,149.434
C01415=1117.452,71.105,-55.395,179.996,7.596,149.433
C01416=1117.456,70.855,-55.378,179.994,7.592,149.433
C01417=1117.461,70.606,-55.360,179.993,7.588,149.432
C01418=1117.466,70.356,-55.343,179.991,7.584,149.432
C01419=1117.470,70.107,-55.325,179.990,7.580,149.431
C01420=1117.476,69.858,-55.308,179.989,7.576,149.431
C01421=1117.481,69.609,-55.290,179.987,7.572,149.430
C01422=1117.486,69.360,-55.274,179.986,7.568,149.430
C01423=1117.491,69.110,-55.256,179.984,7.564,149.429
C01424=1117.496,68.861,-55.238,179.983,7.560,149.429
C01425=1117.500,68.612,-55.221,179.982,7.556,149.428
C01426=1117.505,68.362,-55.204,179.980,7.552,149.428
C01427=1117.510,68.112,-55.187,179.979,7.548,149.427
C01428=1117.515,67.863,-55.169,179.978,7.545,149.427
C01429=1117.520,67.614,-55.152,179.976,7.541,149.426
C01430=1117.526,67.364,-55.135,179.975,7.537,149.426
C01431=1117.530,67.116,-55.118,179.974,7.532,149.425
C01432=1117.535,66.866,-55.100,179.972,7.529,149.425
C01433=1117.539,66.617,-55.083,179.971,7.525,149.424
C01434=1117.544,66.367,-55.066,179.970,7.520,149.424
C01435=1117.550,66.117,-55.048,179.968,7.516,149.423
C01436=1117.554,65.868,-55.032,179.966,7.512,149.423
C01437=1117.560,65.619,-55.014,179.965,7.508,149.422
C01438=1117.564,65.370,-54.997,179.964,7.504,149.422
C01439=1117.569,65.120,-54.980,179.963,7.501,149.421
C01440=1117.573,64.871,-54.963,179.962,7.497,149.421
C01441=1117.579,64.621,-54.946,179.960,7.493,149.420
C01442=1117.584,64.373,-54.929,179.959,7.489,149.420
C01443=1117.589,64.123,-54.912,179.957,7.485,149.419
C01444=1117.593,63.874,-54.895,179.956,7.481,149.419
C01445=1117.598,63.624,-54.877,179.955,7.477,149.418
C01446=1117.603,63.375,-54.861,179.953,7.473,149.418
C01447=1117.609,63.126,-54.844,179.952,7.469,149.417
C01448=1117.612,62.911,-54.829,179.951,7.466,149.417
C01449=1117.617,62.697,-54.815,179.950,7.463,149.416
C01450=1117.620,62.482,-54.800,179.948,7.459,149.416
C01451=1117.625,62.268,-54.786,179.948,7.455,149.415
C01452=1117.629,62.053,-54.771,179.947,7.452,149.415
C01453=1117.634,61.839,-54.756,179.945,7.448,149.414
C01454=1117.637,61.624,-54.742,179.944,7.445,149.414
C01455=1117.642,61.410,-54.727,179.943,7.442,149.414
C01456=1117.647,61.161,-54.710,179.942,7.438,149.413
C01457=1117.652,60.911,-54.693,179.941,7.434,149.412
C01458=1117.657,60.662,-54.676,179.939,7.430,149.412
C01459=1117.662,60.412,-54.659,179.938,7.426,149.412
C01460=1117.667,60.163,-54.643,179.936,7.422,149.411
C01461=1117.671,59.913,-54.626,179.935,7.418,149.411
C01462=1117.677,59.664,-54.609,179.934,7.413,149.410
C01463=1117.681,59.415,-54.592,179.932,7.409,149.409
C01464=1117.686,59.165,-54.575,179.931,7.405,149.409
C01465=1117.692,58.916,-54.559,179.930,7.402,149.408
C01466=1117.696,58.667,-54.542,179.929,7.398,149.408
C01467=1117.701,58.417,-54.525,179.928,7.394,149.407
C01468=1117.706,58.168,-54.508,179.926,7.390,149.407
C01469=1117.711,57.918,-54.492,179.925,7.386,149.406
C01470=1117.716,57.669,-54.475,179.923,7.382,149.406
C01471=1117.721,57.420,-54.458,179.922,7.377,149.405
C01472=1117.726,57.170,-54.442,179.921,7.373,149.405
C01473=1117.731,56.921,-54.424,179.920,7.369,149.404
C01474=1117.736,56.672,-54.408,179.919,7.366,149.404
C01475=1117.740,56.422,-54.391,179.917,7.362,149.403
C01476=1117.746,56.173,-54.374,179.916,7.358,149.403
C01477=1117.751,55.923,-54.358,179.915,7.354,149.402
C01478=1117.755,55.674,-54.342,179.913,7.350,149.401
C01479=1117.760,55.424,-54.325,179.912,7.345,149.401
C01480=1117.766,55.175,-54.308,179.911,7.341,149.400
C01481=1117.770,54.926,-54.292,179.910,7.337,149.400
C01482=1117.775,54.676,-54.275,179.908,7.333,149.399
C01483=1117.780,54.427,-54.259,179.908,7.330,149.399
C01484=1117.785,54.177,-54.242,179.906,7.326,149.398
C01485=1117.790,53.928,-54.226,179.905,7.322,149.398
C01486=1117.795,53.679,-54.209,179.903,7.318,149.397
C01487=1117.799,53.429,-54.192,179.902,7.313,149.396
C01488=1117.806,53.179,-54.176,179.901,7.309,149.396
C01489=1117.810,52.930,-54.160,179.900,7.305,149.395
C01490=1117.815,52.681,-54.143,179.898,7.301,149.395
C01491=1117.820,52.432,-54.127,179.898,7.298,149.394
C01492=1117.825,52.182,-54.111,179.896,7.293,149.394
C01493=1117.830,51.933,-54.094,179.895,7.289,149.393
C01494=1117.835,51.684,-54.077,179.894,7.285,149.393
C01495=1117.840,51.434,-54.061,179.892,7.281,149.392
C01496=1117.845,51.184,-54.045,179.891,7.277,149.392
C01497=1117.850,50.935,-54.028,179.890,7.273,149.391
C01498=1117.854,50.685,-54.013,179.889,7.269,149.390
C01499=1117.859,50.436,-53.996,179.887,7.264,149.390
C01500=1117.865,50.187,-53.979,179.887,7.261,149.389
C01501=1117.870,49.937,-53.963,179.885,7.257,149.389
C01502=1117.875,49.688,-53.947,179.884,7.253,149.388
C01503=1117.880,49.439,-53.930,179.883,7.249,149.388
C01504=1117.883,49.224,-53.916,179.882,7.246,149.387
C01505=1117.888,49.010,-53.903,179.881,7.241,149.387
C01506=1117.892,48.795,-53.889,179.880,7.238,149.386
C01507=1117.897,48.581,-53.875,179.879,7.235,149.386
C01508=1117.901,48.366,-53.861,179.877,7.231,149.385
C01509=1117.905,48.151,-53.847,179.877,7.228,149.385
C01510=1117.909,47.937,-53.833,179.876,7.225,149.384
C01511=1117.913,47.722,-53.819,179.874,7.221,149.384
C01512=1117.918,47.473,-53.803,179.873,7.216,149.383
C01513=1117.923,47.224,-53.787,179.872,7.212,149.383
C01514=1117.928,46.974,-53.771,179.871,7.209,149.382
C01515=1117.933,46.725,-53.755,179.870,7.205,149.381
C01516=1117.938,46.475,-53.739,179.869,7.201,149.381
C01517=1117.943,46.226,-53.723,179.868,7.196,149.380
C01518=1117.948,45.976,-53.707,179.867,7.192,149.380
C01519=1117.953,45.727,-53.690,179.865,7.188,149.379
C01520=1117.958,45.477,-53.674,179.864,7.184,149.379
C01521=1117.963,45.228,-53.658,179.863,7.180,149.378
C01522=1117.968,44.978,-53.642,179.862,7.176,149.377
C01523=1117.973,44.729,-53.627,179.861,7.172,149.377
C01524=1117.978,44.480,-53.610,179.860,7.168,149.376
C01525=1117.983,44.230,-53.594,179.859,7.164,149.376
C01526=1117.988,43.981,-53.578,179.857,7.160,149.375
C01527=1117.993,43.731,-53.562,179.856,7.155,149.374
C01528=1117.998,43.482,-53.546,179.855,7.151,149.374
C01529=1118.003,43.233,-53.530,179.854,7.147,149.373
C01530=1118.008,42.983,-53.514,179.852,7.143,149.373
C01531=1118.013,42.733,-53.499,179.852,7.139,149.372
C01532=1118.018,42.484,-53.482,179.851,7.135,149.371
C01533=1118.023,42.235,-53.467,179.850,7.131,149.371
C01534=1118.028,41.985,-53.451,179.848,7.127,149.370
C01535=1118.032,41.736,-53.435,179.847,7.122,149.370
C01536=1118.038,41.486,-53.419,179.846,7.118,149.369
C01537=1118.043,41.236,-53.403,179.845,7.114,149.368
C01538=1118.048,40.987,-53.388,179.844,7.109,149.368
C01539=1118.053,40.738,-53.371,179.842,7.106,149.367
C01540=1118.057,40.488,-53.356,179.842,7.102,149.367
C01541=1118.062,40.239,-53.340,179.841,7.098,149.366
C01542=1118.068,39.990,-53.325,179.840,7.093,149.365
C01543=1118.073,39.739,-53.309,179.839,7.089,149.365
C01544=1118.078,39.491,-53.293,179.837,7.085,149.364
C01545=1118.083,39.241,-53.277,179.836,7.081,149.364
C01546=1118.087,38.991,-53.262,179.835,7.077,149.363
C01547=1118.093,38.742,-53.246,179.834,7.072,149.362
C01548=1118.098,38.493,-53.230,179.833,7.068,149.362
C01549=1118.103,38.243,-53.215,179.832,7.064,149.361
C01550=1118.107,37.994,-53.199,179.831,7.060,149.360
C01551=1118.112,37.745,-53.183,179.830,7.056,149.360
C01552=1118.118,37.495,-53.168,179.829,7.052,149.359
C01553=1118.123,37.245,-53.152,179.828,7.048,149.359
C01554=1118.128,36.996,-53.136,179.827,7.043,149.358
C01555=1118.133,36.747,-53.121,179.826,7.039,149.357
C01556=1118.138,36.497,-53.105,179.824,7.035,149.357
C01557=1118.143,36.247,-53.089,179.823,7.030,149.356
C01558=1118.147,35.998,-53.074,179.822,7.026,149.355
C01559=1118.153,35.749,-53.059,179.822,7.023,149.355
C01560=1118.157,35.534,-53.045,179.820,7.019,149.354
C01561=1118.162,35.319,-53.032,179.820,7.015,149.354
C01562=1118.166,35.105,-53.018,179.819,7.012,149.353
C01563=1118.170,34.889,-53.005,179.818,7.008,149.353
C01564=1118.174,34.675,-52.991,179.817,7.005,149.352
C01565=1118.178,34.460,-52.979,179.816,7.000,149.351
C01566=1118.183,34.246,-52.965,179.815,6.997,149.351
C01567=1118.187,34.031,-52.952,179.815,6.994,149.350
C01568=1118.193,33.782,-52.937,179.813,6.989,149.350
C01569=1118.197,33.533,-52.922,179.812,6.985,149.349
C01570=1118.203,33.283,-52.906,179.811,6.981,149.348
C01571=1118.207,33.033,-52.890,179.810,6.976,149.348
C01572=1118.212,32.784,-52.875,179.809,6.972,149.347
C01573=1118.217,32.535,-52.860,179.808,6.968,149.346
C01574=1118.223,32.285,-52.844,179.807,6.963,149.346
C01575=1118.227,32.036,-52.829,179.806,6.959,149.345
C01576=1118.232,31.786,-52.813,179.806,6.956,149.345
C01577=1118.237,31.537,-52.798,179.805,6.951,149.344
C01578=1118.243,31.287,-52.783,179.803,6.947,149.343
C01579=1118.248,31.038,-52.768,179.802,6.943,149.343
C01580=1118.253,30.788,-52.753,179.801,6.938,149.342
C01581=1118.258,30.539,-52.737,179.800,6.934,149.341
C01582=1118.262,30.289,-52.722,179.799,6.930,149.341
C01583=1118.267,30.040,-52.706,179.798,6.925,149.340
C01584=1118.272,29.790,-52.692,179.797,6.921,149.339
C01585=1118.278,29.541,-52.676,179.796,6.917,149.339
C01586=1118.282,29.292,-52.661,179.795,6.912,149.338
C01587=1118.288,29.042,-52.646,179.795,6.909,149.337
C01588=1118.293,28.793,-52.631,179.794,6.904,149.336
C01589=1118.297,28.542,-52.615,179.793,6.900,149.336
C01590=1118.302,28.293,-52.600,179.792,6.896,149.335
C01591=1118.308,28.044,-52.585,179.791,6.891,149.335
C01592=1118.312,27.794,-52.571,179.790,6.887,149.334
C01593=1118.318,27.545,-52.555,179.789,6.883,149.333
C01594=1118.323,27.296,-52.540,179.788,6.878,149.333
C01595=1118.328,27.046,-52.525,179.787,6.874,149.332
C01596=1118.333,26.797,-52.510,179.786,6.869,149.331
C01597=1118.338,26.547,-52.495,179.785,6.865,149.330
C01598=1118.343,26.298,-52.480,179.784,6.861,149.330
C01599=1118.347,26.048,-52.465,179.783,6.856,149.329
C01600=1118.353,25.798,-52.449,179.782,6.853,149.328
C01601=1118.358,25.549,-52.435,179.782,6.848,149.328
C01602=1118.363,25.299,-52.419,179.781,6.844,149.327
C01603=1118.368,25.050,-52.404,179.780,6.840,149.326
C01604=1118.373,24.800,-52.390,179.779,6.835,149.326
C01605=1118.378,24.551,-52.375,179.778,6.831,149.325
C01606=1118.383,24.301,-52.360,179.777,6.826,149.324
C01607=1118.388,24.052,-52.345,179.776,6.822,149.323
C01608=1118.393,23.802,-52.330,179.775,6.818,149.323
C01609=1118.398,23.553,-52.315,179.774,6.813,149.322
C01610=1118.403,23.304,-52.300,179.773,6.809,149.321
C01611=1118.408,23.054,-52.286,179.772,6.804,149.321
C01612=1118.413,22.805,-52.271,179.771,6.800,149.320
C01613=1118.419,22.555,-52.256,179.771,6.795,149.319
C01614=1118.423,22.306,-52.241,179.770,6.791,149.318
C01615=1118.428,22.056,-52.226,179.769,6.787,149.318
C01616=1118.433,21.841,-52.213,179.768,6.783,149.317
C01617=1118.437,21.626,-52.200,179.768,6.780,149.316
C01618=1118.441,21.412,-52.188,179.767,6.775,149.316
C01619=1118.446,21.197,-52.175,179.766,6.772,149.315
C01620=1118.450,20.982,-52.163,179.765,6.767,149.314
C01621=1118.454,20.767,-52.150,179.765,6.764,149.314
C01622=1118.459,20.553,-52.138,179.764,6.761,149.313
C01623=1118.463,20.338,-52.125,179.763,6.756,149.313
C01624=1118.468,20.089,-52.110,179.762,6.752,149.312
C01625=1118.473,19.839,-52.095,179.761,6.747,149.311
C01626=1118.479,19.589,-52.081,179.760,6.743,149.311
C01627=1118.483,19.340,-52.066,179.760,6.738,149.310
C01628=1118.488,19.090,-52.051,179.759,6.734,149.309
C01629=1118.493,18.841,-52.037,179.758,6.729,149.308
C01630=1118.499,18.591,-52.021,179.758,6.726,149.307
C01631=1118.504,18.342,-52.007,179.757,6.721,149.307
C01632=1118.509,18.092,-51.993,179.756,6.717,149.306
C01633=1118.513,17.843,-51.978,179.755,6.712,149.305
C01634=1118.518,17.593,-51.964,179.754,6.708,149.304
C01635=1118.524,17.343,-51.949,179.753,6.703,149.304
C01636=1118.529,17.095,-51.934,179.753,6.699,149.303
C01637=1118.534,16.845,-51.920,179.752,6.694,149.302
C01638=1118.539,16.595,-51.906,179.751,6.690,149.301
C01639=1118.544,16.346,-51.891,179.750,6.685,149.301
C01640=1118.549,16.097,-51.876,179.750,6.681,149.300
C01641=1118.554,15.846,-51.861,179.749,6.676,149.299
C01642=1118.559,15.597,-51.847,179.748,6.672,149.298
C01643=1118.564,15.347,-51.833,179.747,6.667,149.298
C01644=1118.569,15.098,-51.818,179.746,6.663,149.297
C01645=1118.574,14.849,-51.804,179.745,6.658,149.296
C01646=1118.579,14.599,-51.790,179.745,6.654,149.295
C01647=1118.584,14.350,-51.775,179.744,6.649,149.294
C01648=1118.589,14.100,-51.761,179.743,6.644,149.294
C01649=1118.594,13.850,-51.747,179.743,6.640,149.293
C01650=1118.600,13.601,-51.731,179.742,6.635,149.292
C01651=1118.605,13.351,-51.717,179.741,6.631,149.291
C01652=1118.610,13.102,-51.703,179.741,6.626,149.290
C01653=1118.615,12.852,-51.689,179.740,6.622,149.290
C01654=1118.620,12.603,-51.674,179.739,6.617,149.289
C01655=1118.625,12.353,-51.660,179.738,6.613,149.288
C01656=1118.630,12.103,-51.646,179.737,6.608,149.287
C01657=1118.636,11.854,-51.632,179.737,6.603,149.286
C01658=1118.640,11.604,-51.618,179.736,6.599,149.286
C01659=1118.645,11.355,-51.603,179.735,6.594,149.285
C01660=1118.650,11.106,-51.588,179.735,6.589,149.284
C01661=1118.655,10.856,-51.574,179.734,6.585,149.283
C01662=1118.661,10.607,-51.560,179.733,6.580,149.282
C01663=1118.666,10.357,-51.546,179.733,6.576,149.282
C01664=1118.670,10.107,-51.532,179.732,6.571,149.281
C01665=1118.675,9.858,-51.517,179.731,6.567,149.280
C01666=1118.680,9.608,-51.503,179.730,6.562,149.279
C01667=1118.686,9.359,-51.489,179.730,6.557,149.278
C01668=1118.691,9.109,-51.475,179.729,6.553,149.277
C01669=1118.696,8.860,-51.461,179.728,6.548,149.277
C01670=1118.701,8.610,-51.446,179.728,6.544,149.276
C01671=1118.707,8.360,-51.433,179.727,6.539,149.275
C01672=1118.711,8.146,-51.421,179.726,6.534,149.274
C01673=1118.714,7.931,-51.408,179.726,6.531,149.273
C01674=1118.719,7.715,-51.396,179.726,6.527,149.273
C01675=1118.724,7.502,-51.384,179.725,6.523,149.272
C01676=1118.728,7.286,-51.372,179.725,6.519,149.271
C01677=1118.732,7.072,-51.360,179.725,6.515,149.271
C01678=1118.737,6.857,-51.348,179.723,6.511,149.270
C01679=1118.741,6.642,-51.336,179.724,6.507,149.269
C01680=1118.746,6.392,-51.322,179.723,6.502,149.268
C01681=1118.751,6.142,-51.308,179.722,6.498,149.267
C01682=1118.756,5.893,-51.295,179.722,6.494,149.267
C01683=1118.761,5.644,-51.280,179.722,6.489,149.266
C01684=1118.766,5.394,-51.266,179.721,6.485,149.265
C01685=1118.772,5.145,-51.252,179.720,6.480,149.264
C01686=1118.777,4.895,-51.239,179.720,6.475,149.263
C01687=1118.782,4.645,-51.224,179.719,6.471,149.262
C01688=1118.787,4.396,-51.210,179.718,6.466,149.262
C01689=1118.792,4.146,-51.197,179.718,6.462,149.261
C01690=1118.797,3.897,-51.182,179.718,6.457,149.260
C01691=1118.803,3.647,-51.169,179.717,6.453,149.259
C01692=1118.807,3.397,-51.155,179.716,6.448,149.258
C01693=1118.812,3.148,-51.141,179.716,6.444,149.257
C01694=1118.817,2.899,-51.127,179.715,6.439,149.256
C01695=1118.822,2.649,-51.114,179.715,6.434,149.256
C01696=1118.827,2.399,-51.099,179.714,6.431,149.255
C01697=1118.833,2.150,-51.086,179.714,6.426,149.254
C01698=1118.838,1.900,-51.073,179.713,6.421,149.253
C01699=1118.842,1.650,-51.058,179.713,6.417,149.252
C01700=1118.848,1.401,-51.044,179.712,6.412,149.251
C01701=1118.853,1.151,-51.031,179.711,6.408,149.251
C01702=1118.859,0.902,-51.017,179.711,6.403,149.250
C01703=1118.863,0.652,-51.003,179.711,6.399,149.249
C01704=1118.868,0.402,-50.990,179.710,6.394,149.248
C01705=1118.874,0.153,-50.976,179.709,6.390,149.247
C01706=1118.878,-0.096,-50.962,179.709,6.385,149.246
C01707=1118.884,-0.346,-50.949,179.708,6.380,149.246
C01708=1118.889,-0.596,-50.935,179.707,6.376,149.245
C01709=1118.894,-0.845,-50.920,179.707,6.371,149.244
C01710=1118.899,-1.095,-50.908,179.706,6.367,149.243
C01711=1118.904,-1.344,-50.893,179.706,6.363,149.242
C01712=1118.910,-1.594,-50.880,179.705,6.358,149.242
C01713=1118.914,-1.843,-50.867,179.705,6.354,149.241
C01714=1118.920,-2.093,-50.853,179.704,6.349,149.240
C01715=1118.925,-2.343,-50.839,179.704,6.344,149.239
C01716=1118.929,-2.593,-50.826,179.703,6.340,149.238
C01717=1118.935,-2.842,-50.812,179.702,6.335,149.237
C01718=1118.940,-3.092,-50.799,179.702,6.330,149.237
C01719=1118.945,-3.341,-50.785,179.701,6.326,149.236
C01720=1118.950,-3.591,-50.772,179.701,6.322,149.235
C01721=1118.955,-3.840,-50.759,179.700,6.317,149.234
C01722=1118.960,-4.090,-50.745,179.699,6.313,149.233
C01723=1118.966,-4.339,-50.731,179.699,6.308,149.233
C01724=1118.970,-4.589,-50.718,179.698,6.304,149.232
C01725=1118.976,-4.838,-50.704,179.698,6.299,149.231
C01726=1118.980,-5.088,-50.691,179.697,6.295,149.230
C01727=1118.986,-5.337,-50.677,179.696,6.290,149.229
C01728=1118.990,-5.552,-50.666,179.696,6.286,149.229
C01729=1118.995,-5.767,-50.654,179.695,6.283,149.228
C01730=1118.999,-5.982,-50.643,179.694,6.278,149.227
C01731=1119.003,-6.198,-50.631,179.694,6.275,149.226
C01732=1119.008,-6.412,-50.620,179.693,6.270,149.226
C01733=1119.012,-6.627,-50.608,179.693,6.267,149.225
C01734=1119.017,-6.842,-50.597,179.693,6.263,149.224
C01735=1119.021,-7.057,-50.585,179.692,6.259,149.224
C01736=1119.026,-7.306,-50.572,179.691,6.254,149.223
C01737=1119.031,-7.556,-50.558,179.691,6.249,149.222
C01738=1119.036,-7.805,-50.545,179.690,6.246,149.221
C01739=1119.042,-8.056,-50.532,179.690,6.241,149.220
C01740=1119.046,-8.305,-50.519,179.689,6.236,149.219
C01741=1119.052,-8.554,-50.505,179.689,6.232,149.219
C01742=1119.057,-8.804,-50.492,179.688,6.227,149.218
C01743=1119.062,-9.053,-50.478,179.687,6.223,149.217
C01744=1119.067,-9.303,-50.466,179.687,6.218,149.216
C01745=1119.073,-9.553,-50.452,179.686,6.213,149.215
C01746=1119.077,-9.803,-50.439,179.685,6.209,149.215
C01747=1119.083,-10.052,-50.425,179.685,6.204,149.214
C01748=1119.088,-10.301,-50.413,179.684,6.200,149.213
C01749=1119.093,-10.551,-50.400,179.683,6.195,149.212
C01750=1119.098,-10.801,-50.387,179.683,6.190,149.211
C01751=1119.103,-11.051,-50.374,179.682,6.186,149.211
C01752=1119.108,-11.300,-50.360,179.681,6.181,149.210
C01753=1119.113,-11.550,-50.347,179.681,6.176,149.209
C01754=1119.119,-11.799,-50.334,179.680,6.172,149.208
C01755=1119.124,-12.049,-50.321,179.679,6.167,149.207
C01756=1119.129,-12.299,-50.308,179.679,6.163,149.206
C01757=1119.134,-12.548,-50.294,179.678,6.158,149.205
C01758=1119.139,-12.797,-50.282,179.677,6.154,149.205
C01759=1119.144,-13.047,-50.269,179.677,6.149,149.204
C01760=1119.150,-13.297,-50.255,179.676,6.144,149.203
C01761=1119.155,-13.546,-50.243,179.676,6.139,149.202
C01762=1119.159,-13.796,-50.230,179.675,6.135,149.201
C01763=1119.165,-14.046,-50.217,179.674,6.130,149.201
C01764=1119.170,-14.296,-50.204,179.674,6.126,149.200
C01765=1119.175,-14.545,-50.191,179.673,6.121,149.199
C01766=1119.181,-14.795,-50.178,179.672,6.117,149.198
C01767=1119.185,-15.044,-50.164,179.672,6.112,149.197
C01768=1119.190,-15.293,-50.152,179.671,6.107,149.196
C01769=1119.196,-15.543,-50.138,179.670,6.103,149.196
C01770=1119.201,-15.792,-50.126,179.670,6.098,149.195
C01771=1119.205,-16.042,-50.113,179.669,6.093,149.194
C01772=1119.211,-16.292,-50.100,179.669,6.089,149.193
C01773=1119.216,-16.541,-50.087,179.668,6.084,149.192
C01774=1119.221,-16.791,-50.074,179.667,6.079,149.191
C01775=1119.226,-17.041,-50.061,179.667,6.075,149.191
C01776=1119.232,-17.290,-50.048,179.666,6.070,149.190
C01777=1119.236,-17.540,-50.035,179.666,6.065,149.189
C01778=1119.242,-17.790,-50.023,179.665,6.061,149.188
C01779=1119.247,-18.040,-50.011,179.664,6.056,149.187
C01780=1119.253,-18.289,-49.998,179.664,6.051,149.186
C01781=1119.257,-18.539,-49.985,179.663,6.047,149.185
C01782=1119.263,-18.789,-49.972,179.662,6.042,149.185
C01783=1119.268,-19.038,-49.959,179.662,6.038,149.184
C01784=1119.272,-19.253,-49.948,179.661,6.033,149.183
C01785=1119.277,-19.468,-49.937,179.661,6.029,149.182
C01786=1119.281,-19.683,-49.926,179.660,6.025,149.182
C01787=1119.285,-19.898,-49.915,179.660,6.021,149.181
C01788=1119.290,-20.113,-49.904,179.659,6.017,149.180
C01789=1119.295,-20.328,-49.894,179.659,6.013,149.179
C01790=1119.299,-20.543,-49.882,179.658,6.009,149.179
C01791=1119.304,-20.758,-49.872,179.657,6.004,149.178
C01792=1119.309,-21.008,-49.859,179.657,5.999,149.177
C01793=1119.313,-21.258,-49.846,179.656,5.995,149.176
C01794=1119.319,-21.507,-49.834,179.656,5.990,149.175
C01795=1119.324,-21.756,-49.821,179.655,5.986,149.174
C01796=1119.329,-22.006,-49.809,179.655,5.981,149.174
C01797=1119.335,-22.256,-49.796,179.654,5.976,149.173
C01798=1119.340,-22.505,-49.783,179.654,5.971,149.172
C01799=1119.345,-22.755,-49.770,179.653,5.966,149.171
C01800=1119.350,-23.005,-49.759,179.652,5.961,149.170
C01801=1119.355,-23.254,-49.746,179.651,5.957,149.169
C01802=1119.360,-23.504,-49.733,179.651,5.952,149.168
C01803=1119.365,-23.753,-49.721,179.650,5.947,149.167
C01804=1119.371,-24.003,-49.709,179.650,5.943,149.167
C01805=1119.375,-24.253,-49.696,179.649,5.937,149.166
C01806=1119.380,-24.502,-49.683,179.648,5.932,149.165
C01807=1119.386,-24.752,-49.671,179.648,5.928,149.164
C01808=1119.391,-25.002,-49.659,179.647,5.923,149.163
C01809=1119.396,-25.251,-49.646,179.647,5.918,149.162
C01810=1119.402,-25.501,-49.634,179.646,5.913,149.161
C01811=1119.407,-25.750,-49.622,179.645,5.908,149.160
C01812=1119.411,-26.000,-49.609,179.645,5.904,149.159
C01813=1119.417,-26.250,-49.597,179.646,5.900,149.158
